			IF fbTimer.Q 
			THEN
				fbTimer(IN := FALSE); 			
				eReadDiagObjState := eCycleDiagObj_Done;
			END_IF

			
		eCycleDiagObj_Done				:	(* Done *)

			eReadDiagObjState := eCycleDiagObj_Init;

			
		eCycleDiagObj_Error			:	(* Error detected *)

			bReadDiagObjError := TRUE;
		
			IF bReadDiagObjReset
			THEN
				bReadDiagObjError 		:= FALSE;
				fbEcCoeSdoRead(bExecute := FALSE);
				eReadDiagObjErrStep 	:= E_TsCycleDiagObj.eCycleDiagObj_NoError;
				eReadDiagObjState 		:= eCycleDiagObj_Init;
			END_IF

	ELSE
		
		eReadDiagObjState := eCycleDiagObj_Init;
		
	END_CASE

	bTempWarning := stSlaveTemp.nInternalTemperature1 >= nWarningLevelTemp1 
						OR stSlaveTemp.nInternalTemperature2 >= nWarningLevelTemp2;

(* End *)
END_ACTION

ACTION act_Signals:
(* Evaluate the input and output signals *)

	IF nEcSlaveState.3 (* Slave in operational state *)
	THEN
	
		(* OP -> transfer the signal states *)
		stSignalStatusMC1.bSafeTorqueOff_STO 					:= stInfoData.nInSafeDataByte1.0;
		stSignalStatusMC1.bSafeSpeedMonitor_SSM_1 				:= stInfoData.nInSafeDataByte1.1;
		stSignalStatusMC1.bSafeSpeedMonitor_SSM_2 				:= stInfoData.nInSafeDataByte1.2;
		stSignalStatusMC1.bSafeOperatingStop_SOS_1	 			:= stInfoData.nInSafeDataByte1.3;
		stSignalStatusMC1.bSafeSpeedRange_SSR_1 				:= stInfoData.nInSafeDataByte1.4;
		stSignalStatusMC1.bSafeDirectionPositive_SDIp 			:= stInfoData.nInSafeDataByte1.5;
		stSignalStatusMC1.bSafeDirectionNegative_SDIn 			:= stInfoData.nInSafeDataByte1.6;
		stSignalStatusMC1.bErrorAcknowledge_ErrAck 				:= stInfoData.nInSafeDataByte1.7;
		stSignalStatusMC1.bNotInUseBit8 						:= stInfoData.nInSafeDataByte2.0;
		stSignalStatusMC1.bNotInUseBit9 						:= stInfoData.nInSafeDataByte2.1;
		stSignalStatusMC1.bNotInUseBit10						:= stInfoData.nInSafeDataByte2.2;
		stSignalStatusMC1.bNotInUseBit11						:= stInfoData.nInSafeDataByte2.3;
		stSignalStatusMC1.bNotInUseBit12						:= stInfoData.nInSafeDataByte2.4;
		stSignalStatusMC1.bNotInUseBit13						:= stInfoData.nInSafeDataByte2.5;
		stSignalStatusMC1.bNotInUseBit14						:= stInfoData.nInSafeDataByte2.6;
		stSignalStatusMC1.bNotInUseBit15						:= stInfoData.nInSafeDataByte2.7;
		
		stSignalStatusMC2.bSafeTorqueOff_STO 					:= stInfoData.nInSafeDataByte3.0;
		stSignalStatusMC2.bSafeSpeedMonitor_SSM_1 				:= stInfoData.nInSafeDataByte3.1;
		stSignalStatusMC2.bSafeSpeedMonitor_SSM_2 				:= stInfoData.nInSafeDataByte3.2;
		stSignalStatusMC2.bSafeOperatingStop_SOS_1 				:= stInfoData.nInSafeDataByte3.3;
		stSignalStatusMC2.bSafeSpeedRange_SSR_1 				:= stInfoData.nInSafeDataByte3.4;
		stSignalStatusMC2.bSafeDirectionPositive_SDIp 			:= stInfoData.nInSafeDataByte3.5;
		stSignalStatusMC2.bSafeDirectionNegative_SDIn		 	:= stInfoData.nInSafeDataByte3.6;
		stSignalStatusMC2.bErrorAcknowledge_ErrAck 				:= stInfoData.nInSafeDataByte3.7;
		stSignalStatusMC2.bNotInUseBit8 						:= stInfoData.nInSafeDataByte4.0;
		stSignalStatusMC2.bNotInUseBit9 						:= stInfoData.nInSafeDataByte4.1;
		stSignalStatusMC2.bNotInUseBit10						:= stInfoData.nInSafeDataByte4.2;
		stSignalStatusMC2.bNotInUseBit11						:= stInfoData.nInSafeDataByte4.3;
		stSignalStatusMC2.bNotInUseBit12						:= stInfoData.nInSafeDataByte4.4;
		stSignalStatusMC2.bNotInUseBit13						:= stInfoData.nInSafeDataByte4.5;
		stSignalStatusMC2.bNotInUseBit14						:= stInfoData.nInSafeDataByte4.6;
		stSignalStatusMC2.bNotInUseBit15						:= stInfoData.nInSafeDataByte4.7;
		
		stSignalControlStatusMC1.bSafeTorqueOff_STO 			:= stInfoData.nOutSafeDataByte1.0;
		stSignalControlStatusMC1.bSafeStop1_SS1_1 				:= stInfoData.nOutSafeDataByte1.1;
		stSignalControlStatusMC1.bSafeStop2_SS2_1 				:= stInfoData.nOutSafeDataByte1.2;
		stSignalControlStatusMC1.bSafeOperatingStop_SOS_1 		:= stInfoData.nOutSafeDataByte1.3;
		stSignalControlStatusMC1.bSafeSpeedRange_SSR_1 			:= stInfoData.nOutSafeDataByte1.4;
		stSignalControlStatusMC1.bSafeDirectionPositive_SDIp 	:= stInfoData.nOutSafeDataByte1.5;
		stSignalControlStatusMC1.bSafeDirectionNegative_SDIn 	:= stInfoData.nOutSafeDataByte1.6;
		stSignalControlStatusMC1.bErrorAcknowledge_ErrAck 		:= stInfoData.nOutSafeDataByte1.7;
		stSignalControlStatusMC1.bNotInUseBit8 					:= stInfoData.nOutSafeDataByte2.0;
		stSignalControlStatusMC1.bNotInUseBit9 					:= stInfoData.nOutSafeDataByte2.1;
		stSignalControlStatusMC1.bNotInUseBit10					:= stInfoData.nOutSafeDataByte2.2;
		stSignalControlStatusMC1.bNotInUseBit11					:= stInfoData.nOutSafeDataByte2.3;
		stSignalControlStatusMC1.bNotInUseBit12					:= stInfoData.nOutSafeDataByte2.4;
		stSignalControlStatusMC1.bNotInUseBit13					:= stInfoData.nOutSafeDataByte2.5;
		stSignalControlStatusMC1.bNotInUseBit14					:= stInfoData.nOutSafeDataByte2.6;
		stSignalControlStatusMC1.bNotInUseBit15					:= stInfoData.nOutSafeDataByte2.7;

		stSignalControlStatusMC2.bSafeTorqueOff_STO 			:= stInfoData.nOutSafeDataByte3.0;
		stSignalControlStatusMC2.bSafeStop1_SS1_1 				:= stInfoData.nOutSafeDataByte3.1;
		stSignalControlStatusMC2.bSafeStop2_SS2_1 				:= stInfoData.nOutSafeDataByte3.2;
		stSignalControlStatusMC2.bSafeOperatingStop_SOS_1 		:= stInfoData.nOutSafeDataByte3.3;
		stSignalControlStatusMC2.bSafeSpeedRange_SSR_1 			:= stInfoData.nOutSafeDataByte3.4;
		stSignalControlStatusMC2.bSafeDirectionPositive_SDIp 	:= stInfoData.nOutSafeDataByte3.5;
		stSignalControlStatusMC2.bSafeDirectionNegative_SDIn 	:= stInfoData.nOutSafeDataByte3.6;
		stSignalControlStatusMC2.bErrorAcknowledge_ErrAck 		:= stInfoData.nOutSafeDataByte3.7;
		stSignalControlStatusMC2.bNotInUseBit8 					:= stInfoData.nOutSafeDataByte4.0;
		stSignalControlStatusMC2.bNotInUseBit9 					:= stInfoData.nOutSafeDataByte4.1;
		stSignalControlStatusMC2.bNotInUseBit10					:= stInfoData.nOutSafeDataByte4.2;
		stSignalControlStatusMC2.bNotInUseBit11					:= stInfoData.nOutSafeDataByte4.3;
		stSignalControlStatusMC2.bNotInUseBit12					:= stInfoData.nOutSafeDataByte4.4;
		stSignalControlStatusMC2.bNotInUseBit13					:= stInfoData.nOutSafeDataByte4.5;
		stSignalControlStatusMC2.bNotInUseBit14					:= stInfoData.nOutSafeDataByte4.6;
		stSignalControlStatusMC2.bNotInUseBit15					:= stInfoData.nOutSafeDataByte4.7;
		
	ELSE
		
		(* Error -> clear the signal states *)
		stSignalStatusMC1.bSafeTorqueOff_STO 					:= FALSE;
		stSignalStatusMC1.bSafeSpeedMonitor_SSM_1 				:= FALSE;
		stSignalStatusMC1.bSafeSpeedMonitor_SSM_2 				:= FALSE;
		stSignalStatusMC1.bSafeOperatingStop_SOS_1	 			:= FALSE;
		stSignalStatusMC1.bSafeSpeedRange_SSR_1 				:= FALSE;
		stSignalStatusMC1.bSafeDirectionPositive_SDIp 			:= FALSE;
		stSignalStatusMC1.bSafeDirectionNegative_SDIn 			:= FALSE;
		stSignalStatusMC1.bErrorAcknowledge_ErrAck 				:= FALSE;
		stSignalStatusMC1.bNotInUseBit8 						:= FALSE;
		stSignalStatusMC1.bNotInUseBit9 						:= FALSE;
		stSignalStatusMC1.bNotInUseBit10						:= FALSE;
		stSignalStatusMC1.bNotInUseBit11						:= FALSE;
		stSignalStatusMC1.bNotInUseBit12						:= FALSE;
		stSignalStatusMC1.bNotInUseBit13						:= FALSE;
		stSignalStatusMC1.bNotInUseBit14						:= FALSE;
		stSignalStatusMC1.bNotInUseBit15						:= FALSE;
		
		stSignalStatusMC2.bSafeTorqueOff_STO 					:= FALSE;
		stSignalStatusMC2.bSafeSpeedMonitor_SSM_1 				:= FALSE;
		stSignalStatusMC2.bSafeSpeedMonitor_SSM_2 				:= FALSE;
		stSignalStatusMC2.bSafeOperatingStop_SOS_1 				:= FALSE;
		stSignalStatusMC2.bSafeSpeedRange_SSR_1 				:= FALSE;
		stSignalStatusMC2.bSafeDirectionPositive_SDIp 			:= FALSE;
		stSignalStatusMC2.bSafeDirectionNegative_SDIn		 	:= FALSE;
		stSignalStatusMC2.bErrorAcknowledge_ErrAck 				:= FALSE;
		stSignalStatusMC2.bNotInUseBit8 						:= FALSE;
		stSignalStatusMC2.bNotInUseBit9 						:= FALSE;
		stSignalStatusMC2.bNotInUseBit10						:= FALSE;
		stSignalStatusMC2.bNotInUseBit11						:= FALSE;
		stSignalStatusMC2.bNotInUseBit12						:= FALSE;
		stSignalStatusMC2.bNotInUseBit13						:= FALSE;
		stSignalStatusMC2.bNotInUseBit14						:= FALSE;
		stSignalStatusMC2.bNotInUseBit15						:= FALSE;
		
		stSignalControlStatusMC1.bSafeTorqueOff_STO 			:= FALSE;
		stSignalControlStatusMC1.bSafeStop1_SS1_1 				:= FALSE;
		stSignalControlStatusMC1.bSafeStop2_SS2_1 				:= FALSE;
		stSignalControlStatusMC1.bSafeOperatingStop_SOS_1 		:= FALSE;
		stSignalControlStatusMC1.bSafeSpeedRange_SSR_1 			:= FALSE;
		stSignalControlStatusMC1.bSafeDirectionPositive_SDIp 	:= FALSE;
		stSignalControlStatusMC1.bSafeDirectionNegative_SDIn 	:= FALSE;
		stSignalControlStatusMC1.bErrorAcknowledge_ErrAck 		:= FALSE;
		stSignalControlStatusMC1.bNotInUseBit8 					:= FALSE;
		stSignalControlStatusMC1.bNotInUseBit9 					:= FALSE;
		stSignalControlStatusMC1.bNotInUseBit10					:= FALSE;
		stSignalControlStatusMC1.bNotInUseBit11					:= FALSE;
		stSignalControlStatusMC1.bNotInUseBit12					:= FALSE;
		stSignalControlStatusMC1.bNotInUseBit13					:= FALSE;
		stSignalControlStatusMC1.bNotInUseBit14					:= FALSE;
		stSignalControlStatusMC1.bNotInUseBit15					:= FALSE;

		stSignalControlStatusMC2.bSafeTorqueOff_STO 			:= FALSE;
		stSignalControlStatusMC2.bSafeStop1_SS1_1 				:= FALSE;
		stSignalControlStatusMC2.bSafeStop2_SS2_1 				:= FALSE;
		stSignalControlStatusMC2.bSafeOperatingStop_SOS_1 		:= FALSE;
		stSignalControlStatusMC2.bSafeSpeedRange_SSR_1 			:= FALSE;
		stSignalControlStatusMC2.bSafeDirectionPositive_SDIp 	:= FALSE;
		stSignalControlStatusMC2.bSafeDirectionNegative_SDIn 	:= FALSE;
		stSignalControlStatusMC2.bErrorAcknowledge_ErrAck 		:= FALSE;
		stSignalControlStatusMC2.bNotInUseBit8 					:= FALSE;
		stSignalControlStatusMC2.bNotInUseBit9 					:= FALSE;
		stSignalControlStatusMC2.bNotInUseBit10					:= FALSE;
		stSignalControlStatusMC2.bNotInUseBit11					:= FALSE;
		stSignalControlStatusMC2.bNotInUseBit12					:= FALSE;
		stSignalControlStatusMC2.bNotInUseBit13					:= FALSE;
		stSignalControlStatusMC2.bNotInUseBit14					:= FALSE;
		stSignalControlStatusMC2.bNotInUseBit15					:= FALSE;

	END_IF

(* End *)
END_ACTION

END_FUNCTION_BLOCK

// ---- POUs/Motion/NCI.TcPOU
PROGRAM NCI
VAR
(* NCI G code stuff *)

	in_stItpToPlc		AT 	%I*:	NCTOPLC_NCICHANNEL_REF;
	out_stPlcToItp		AT	%Q*:	PLCTONC_NCICHANNEL_REF;
	
	bRunNCI				: BOOL;
	bErrorAck			: BOOL;

(*
	g_strProgram:	STRING := 'Hard Disk2\TestIt.nc';	(* USB stick with CE OS *)
*)
	g_strProgram		: STRING := 'C:\btest.nc';

	bNCIExec			: BOOL;
	bNCIBusy			: BOOL := FALSE;
	bNciErr				: BOOL := FALSE;
	nNciErrId			: UDINT := 0;

	nNCI_State			: UDINT := 0;
	nLastState			: UDINT	:= 0;	(* for debugging purposes *)
	fbBuildGrp			: CfgBuildExt3DGroup;
	fbLoadProg			: ItpLoadProgEx;
	fbStart				: ItpStartStopEx;
	
	fbConfirm			: ItpConfirmHsk;
	bConfirm			: BOOL := FALSE;
	
	fbClearGrp			: CfgReconfigGroup;
	fbResetItp			: ItpResetEx2;
	nItpState			: UDINT;

	bPenDown : BOOL;

	fbADSREAD_NciLine	: ADSREAD;
	sGCodeLine			: STRING(254);
	sGCodeLineLast		: STRING(254);
	bReadGcodeLine		: BOOL;
	bItpReset			: BOOL;

	aGCodeLines			: ARRAY[0..9] OF STRING[254];
	iLine				: UINT;
END_VAR

ItpSetOverridePercent(100.0, out_stPlcToItp);

CASE nNCI_State OF
0:
	if bRunNCI then
		nNCI_State := 5;
	END_IF
	
5:
	bNCIBusy	:= TRUE;
	bNciErr	:= FALSE;
	nNciErrId	:= 0;
	nLastState	:= 0;
	nNCI_State 	:= 10;
	FOR iLine := 0 TO 9 DO
			aGCodeLines[iLine]:='';
	END_FOR


10:
	(* build interpolation group *)
	fbBuildGrp(
		bExecute	:= TRUE ,
		nGroupId	:= ItpGetGroupId(sNciToPlc:=in_stItpToPlc),
		nXAxisId	:= stAxis3.NcToPlc.AxisId,
		nYAxisId	:= stAxis4.NcToPlc.AxisId,
		nZAxisId	:= 0,
		nQ1AxisId:= 0,
		nQ2AxisId:= 0,
		nQ3AxisId:= 0,
		nQ4AxisId:= 0,
		nQ5AxisId:= 0,
		tTimeOut:= T#200ms);

	IF NOT fbBuildGrp.bBusy THEN
		fbBuildGrp( bExecute := FALSE );
		IF NOT fbBuildGrp.bErr THEN
			nNCI_State	:= 20;
		ELSE
			(* an error occured *)
			bNciErr		:= TRUE;
			nNciErrId	:= fbBuildGrp.nErrId;
			nLastState	:= nNCI_State;
			nNCI_State	:= 9999;
		END_IF
	END_IF

20:
	(* load part program *)
	fbLoadProg(
		bExecute	:= TRUE,
		sPrg		:= g_strProgram,
		nLength		:= INT_TO_UDINT(LEN(g_strProgram)),
		tTimeOut	:= t#200ms,
		sNciToPlc:= in_stItpToPlc );

	IF NOT fbLoadProg.bBusy THEN
		fbLoadProg( bExecute:=FALSE, sNciToPlc:=in_stItpToPlc );
		IF NOT fbLoadProg.bErr THEN
			nNCI_State	:= 30;
		ELSE
			(* an error occured *)
			bNciErr		:= TRUE;
			nNciErrId	:= fbLoadProg.nErrId;
			nLastState	:= nNCI_State;
			nNCI_State	:= 9999;
		END_IF
	END_IF

30:
	(* wait until interpreter is in ready state *)
	nItpState	:=	ItpGetStateInterpreter( in_stItpToPlc );
	IF nItpState = NCI_INTERPRETER_READY THEN
		(* load part program succeeded *)
		nNCI_State	:= 40;
	ELSIF nItpState = NCI_INTERPRETER_ABORTED THEN
		(* load program failed - probably there is a load time error, e.g. syntax error *)
		(* add error handling here *)
		bNciErr		:= TRUE;
		nNciErrId	:= 4711;	(* substitute with own error code *)
		nLastState	:= nNCI_State;
		nNCI_State	:= 9999;
	END_IF

40:
	(* start part program *)
	fbStart(
		bStart	:= TRUE,
		bStop		:= FALSE,
		tTimeOut	:= t#200ms,
		sNciToPlc:= in_stItpToPlc );

	IF NOT fbStart.bBusy THEN
		fbStart( bStart:=FALSE, sNciToPlc:=in_stItpToPlc );
		IF NOT fbStart.bErr THEN
			nNCI_State	:= 50;
		ELSE
			(* an error occured *)
			bNciErr		:= TRUE;
			nNciErrId	:= fbStart.nErrId;
			nLastState	:= nNCI_State;
			nNCI_State	:= 9999;
		END_IF
	END_IF

50:
	(* check if the part program is really started *)
	(* as long as the part program is active we are not in the ready state *)
	(* if the part program has finished without an error we switch back to the ready state *)
	(* if the program has finished with an error the interpreter is in the aborted state *)
	nItpState	:=	ItpGetStateInterpreter( in_stItpToPlc );
	IF nItpState <> NCI_INTERPRETER_READY THEN
		nNCI_State	:= 60;
		// bReadGcodeLine := TRUE;
	END_IF

60:
	(* Confirmed m-functions *)
	(*
	IF ( ItpIsHskMFunc(in_stItpToPlc) ) THEN
		bConfirm	:= TRUE;
	ELSE
		bConfirm	:= FALSE;
	END_IF

	fbConfirm(
		bExecute:= bConfirm,
		sNciToPlc:= in_stItpToPlc,
		sPlcToNci:= out_stPlcToItp );

	IF NOT fbConfirm.bBusy THEN
		IF fbConfirm.bErr THEN
			(* an error occured *)
			(* this usually can just occur, if a confirmation is triggered without a request *)
			bNCIErr		:= TRUE;
			iNCIErrId	:= fbStart.nErrId;
			iNCILastState	:= iNCIState;
			iNCIState	:= 9999;
		END_IF
	END_IF
	*)

(* code for fast M function with no handshaking - example M100/M101 to trigger 'Pen down' boolean *)
	IF ItpIsFastMFunc(100, in_stItpToPlc ) THEN
		bPenDown:= TRUE;
	ELSE
		bPenDown:= FALSE;
	END_IF

	nItpState	:=	ItpGetStateInterpreter( in_stItpToPlc );
	IF nItpState = NCI_INTERPRETER_READY THEN
		(* part program is finished without an error *)
		nNCI_State	:= 70;
	ELSIF nItpState = NCI_INTERPRETER_ABORTED THEN
		(* a runtime error occured - e.g. a lag distance error occured *)
		bNciErr		:= TRUE;
		nNciErrId	:= ItpGetError(in_stItpToPlc);
		nLastState	:= nNCI_State;
		nNCI_State	:= 9999;
	END_IF

	(* Read executing Gcode lines *)
	fbADSREAD_NciLine(
		NETID:= '',
		PORT:= 500,
		IDXGRP:= 16#2302,
		IDXOFFS:= 16#20000001,
		LEN:= 248,
		DESTADDR:= ADR(sGCodeLine),
		READ:= bReadGcodeLine,
		TMOUT:= t#200ms,
		BUSY=> ,
		ERR=> ,
		ERRID=> );

	IF fbADSREAD_NciLine.BUSY = FALSE THEN
		IF bReadGcodeLine = TRUE THEN
			bReadGcodeLine:=FALSE;
			IF sGCodeLineLast<>sGCodeLine THEN
				// shift table down and add line to top of table
				MEMMOVE(destAddr:= ADR(aGCodeLines[1]), srcAddr:= ADR(aGCodeLines[0]), n:= 254*9);
				aGCodeLines[0]:=sGCodeLine;
				sGCodeLineLast:=sGCodeLine;
			END_IF
		ELSE
			bReadGcodeLine:=TRUE;
		END_IF
	END_IF

70:
	(* clear interpolation group *)
	fbClearGrp(
		bExecute:= TRUE,
		nGroupId:= ItpGetGroupId(sNciToPlc:=in_stItpToPlc),
		tTimeOut:= T#200ms);

	IF NOT fbClearGrp.bBusy THEN
		fbClearGrp(bExecute:= FALSE);
		IF NOT fbClearGrp.bErr THEN
			nNCI_State	:= 100;
		ELSE
			(* an error occured *)
			bNciErr		:= TRUE;
			nNciErrId	:= fbClearGrp.nErrId;
			nLastState	:= nNCI_State;
			nNCI_State	:= 9999;
		END_IF
	END_IF

100:	(* Finished NCI successfully *)
	bNciBusy	:= FALSE;
	fbBuildGrp( bExecute:=FALSE );
	fbLoadProg( bExecute:=FALSE, sNciToPlc:=in_stItpToPlc );
	fbStart( bStart:=FALSE, bStop:=FALSE, sNciToPlc:=in_stItpToPlc );
	fbClearGrp(bExecute:= FALSE);

	bPenDown:= FALSE;
	bReadGcodeLine:=FALSE;

	nNci_State	:= 0;

9999:
	bNCIBusy	:= FALSE;
	fbBuildGrp( bExecute:=FALSE );
	fbLoadProg( bExecute:=FALSE, sNciToPlc:=in_stItpToPlc );
	fbStart( bStart:=FALSE, bStop:=FALSE, sNciToPlc:=in_stItpToPlc );
	fbClearGrp(bExecute:= FALSE);

	bPenDown:= FALSE;
	bReadGcodeLine:=FALSE;

	IF bErrorAck THEN
		nNCI_State	:= 0;
		nNciErrId	:= 0;
	END_IF

END_CASE

END_PROGRAM

// ---- POUs/Motion/CamTable.TcPOU
PROGRAM CamTable
VAR
	bLoadPoints: BOOL;
	bCamInit			: BOOL;

	arCamTable			: ARRAY [0..iNumPts, 0..1] OF LREAL;
	CamTblSelect		: MC_CamTableSelect;
	CamTableRef			: MC_Cam_Ref;
	ST_CamInOptions_V2	: ST_CamInOptions_V2;

	CamIn_v2			: MC_CamIn_V2;
	CamOut				: MC_CamOut;
	bCamIn				: BOOL;

	osrTblSlct			: F_TRIG;
	bPeriodic			: BOOL;

	iInterpType			: UINT :=1;		// start with spline

	iSelX				: INT;			// selected visualization col
	iSelY				: INT;			// selected visualization row 
	
END_VAR

VAR CONSTANT
	iNumPts 			: UDINT := 5;
END_VAR

Cam_Setup();

IF bLoadPoints THEN
	LoadPoints();
	bLoadPoints:=FALSE;
END_IF

IF bCamInit THEN
	Cam_Init();
	bCamInit := FALSE;
END_IF

ACTION Cam_Init:

CamTableRef.pArray := ADR(arCamTable);
CamTableRef.ArraySize := SIZEOF(arCamTable);

CamTableRef.TableType := MC_TABLETYPE_EQUIDISTANT ;

CamTableRef.NoOfRows := iNumPts;
CamTableRef.NoOfColumns := 2;
ST_CamInOptions_V2.CamOperationMode:=CAMOPERATIONMODE_ADDITIVE;


CASE iInterpType OF
0:
	ST_CamInOptions_V2.InterpolationType:=MC_INTERPOLATIONTYPE_LINEAR;
1:
	ST_CamInOptions_V2.InterpolationType:=MC_INTERPOLATIONTYPE_SPLINE;
2:
	ST_CamInOptions_V2.InterpolationType:=MC_INTERPOLATIONTYPE_SLIDINGSPLINE;
END_CASE
END_ACTION

ACTION Cam_Setup:
osrTblSlct(CLK := bCamInit); // F_TRIG
CamIn_v2(
    Master := stAxis3,
    Slave := stAxis4,
    Execute := bCamIn,
    ActivationMode := MC_CAMACTIVATION_INSTANTANEOUS,
    CamTableID := 2,
    Options := ST_CamInOptions_V2); // MC_CamIn_V2
CamTblSelect(
    Execute := NOT CamTblSelect.Done AND osrTblSlct.Q,
    Periodic := bPeriodic,
    CamTableID := 2,
    Master := stAxis3,
    Slave := stAxis4,
    CamTable := CamTableRef); // MC_CamTableSelect
CamOut(Execute := NOT(bCamIn), Slave := stAxis4); // MC_CamOut
END_ACTION

ACTION LoadPoints:
arCamTable[0,0] := 0;
arCamTable[0,1] := 0;

arCamTable[1,0] := 250;
arCamTable[1,1] := 500;

arCamTable[2,0] := 500;
arCamTable[2,1] := 1000;

arCamTable[3,0] := 750;
arCamTable[3,1] := 500;

arCamTable[4,0] := 1000;
arCamTable[4,1] := 0;
END_ACTION

END_PROGRAM

// ---- POUs/Motion/Ext_SP_Gen.TcPOU
PROGRAM Ext_SP_Gen
VAR
	bMstrExtSP			: BOOL;
	ExtSP_Enable		: MC_ExtSetPointGenEnable;
	ExtSP_Disable		: MC_ExtSetPointGenDisable;	

	lrPosCmd			: LREAL;
	lrVeloCmd			: LREAL;
	lrAccelCmd			: LREAL;

	rDeg				: REAL;
	rDegStep			: REAL := 0.1;
	lrSinWave			: LREAL;
	rSinAmp				: REAL := 30.0;
	
	bSinGen				: BOOL;
	bAddSin				: BOOL;

	diDir: DINT := 1;
	
	lrPosInput: LREAL;
END_VAR

IF bSinGen THEN
	rDeg:=rDeg+rDegStep;
	IF rDeg >= 360.0 THEN
		rDeg:=0.0;
	END_IF
END_IF

lrSinWave:=rSinAmp*SIN(rDeg*3.14159/180.0);	// SIN function uses radian input

IF bAddSin THEN
	lrPosCmd:=lrPosInput+lrSinWave;
ELSE
	lrPosCmd:=lrPosInput;
END_IF

MC_ExtSetPointGenFeed(
	lrPosCmd,
	lrVeloCmd,
	lrAccelCmd,
	diDir,
	stAxis3);

ExtSP_Enable(
	Axis:= stAxis3, 
	Execute:= bMstrExtSP, 
	Position:= , 
	PositionType:= POSITIONTYPE_ABSOLUTE, 
	Done=> , 
	Busy=> , 
	Error=> , 
	ErrorID=> , 
	Enabled=> );
	
ExtSP_Disable(
	Axis:= stAxis3, 
	Execute:= NOT(bMstrExtSP), 
	Done=> , 
	Busy=> , 
	Error=> , 
	ErrorID=> , 
	Enabled=> );

END_PROGRAM

// ---- POUs/SampleIEC Languages/MAIN_CFC.TcPOU
PROGRAM MAIN_CFC
VAR
	Timer			: TON;
	fbCFC_SamplePOU : FB_CFC_SamplePOU;

	eOperation		: E_Operation := eOp_Add;
	eOperationPrev	: E_Operation := eOp_Add;
	iResultC		: DINT;
	bZero			: BOOL;
	bPos			: BOOL;
	bNeg			: BOOL;
	bTest			: BOOL;
	tTimerValue		: TIME := T#3S;
END_VAR
VAR // added by the converter: edge detectors and wires of the graphical bodies
    _w1, _w2, _w3 : E_Operation;
END_VAR

bTest := (bZero AND bPos OR bPos XOR bNeg) AND iResultC <= 0 AND Timer.ET > T#500ms OR Timer.ET <= T#500ms;
// Timer
Timer(IN := NOT Timer.Q, PT := tTimerValue); // TON
IF NOT Timer.Q THEN JMP CALLFB; END_IF
// State machine
_w1 := SEL(eOp_Add = eOperation AND Timer.Q, eOperation, eOp_Mul);
eOperation := _w1;
IF _w1 <> eOperationPrev AND _w1 = eOp_Mul THEN JMP CallFB; END_IF
_w2 := SEL(eOp_Sub = eOperation AND Timer.Q, eOperation, eOp_Add);
eOperation := _w2;
IF _w2 <> eOperationPrev AND _w2 = eOp_Add THEN JMP CallFB; END_IF
_w3 := SEL(eOp_Mul = eOperation AND Timer.Q, eOperation, eOp_Sub);
eOperation := _w3;
IF _w3 <> eOperationPrev AND _w3 = eOp_Sub THEN JMP CallFB; END_IF
// FB Call
CallFB: ;
eOperationPrev := eOperation;
fbCFC_SamplePOU(eOperation := eOperation); // FB_CFC_SamplePOU
iResultC := fbCFC_SamplePOU.iResultC;
bZero := fbCFC_SamplePOU.iResultC = 0;
bPos := fbCFC_SamplePOU.iResultC > 0;
bNeg := fbCFC_SamplePOU.iResultC < 0;

END_PROGRAM

// ---- POUs/SampleIEC Languages/FunctionBlocks/FB_CFC_SamplePOU.TcPOU
FUNCTION_BLOCK FB_CFC_SamplePOU
VAR_INPUT
//	eOperation	: INT;
	eOperation	: E_Operation;
END_VAR
VAR_OUTPUT
	iResultC	: DINT;
END_VAR
VAR
	arrDataA	: ARRAY [1..iMax] OF DINT;
	arrDataB	: ARRAY [1..iMax] OF DINT;
	arrDataC	: ARRAY [1..iMax] OF DINT;
	I 			: DINT;
	bInit		: BOOL := TRUE;
END_VAR
VAR CONSTANT
	iMax 		: DINT := 10;
END_VAR
VAR // added by the converter: edge detectors and wires of the graphical bodies
    _w1, _w2, _w4, _w6, _w9 : DINT;
    _w3, _w5, _w8 : ANY;
    _w7 : BOOL;
END_VAR

IF NOT bInit THEN JMP SkipInit; END_IF
bInit := FALSE;
I := 1;
Init: ;
_w1 := iMax - I;
arrDataA[I] := _w1;
arrDataB[I] := _w1 + 1;
_w2 := I + 1;
I := _w2;
IF _w2 <= iMax THEN JMP Init; END_IF
SkipInit: ;
IF eOperation = eOp_Add THEN JMP OP_Add; END_IF
IF eOperation = eOp_Sub THEN JMP OP_Sub; END_IF
IF eOperation = eOp_Mul THEN JMP OP_Mul; END_IF
IF TRUE THEN JMP END; END_IF
OP_Add: ;
iResultC := 0;
I := 1 + 0;
WHILE4_0: ;
IF I > iMax THEN JMP END; END_IF
_w3 := arrDataA[I] + arrDataB[I];
arrDataC[I] := _w3;
iResultC := iResultC + _w3;
_w4 := I + 1;
I := _w4;
IF _w4 >= _w4 THEN JMP WHILE4_0; END_IF
OP_Sub: ;
iResultC := 0;
I := 1 + 0;
Repeat5_0: ;
_w5 := arrDataA[I] - arrDataB[I];
arrDataC[I] := _w5;
iResultC := iResultC + _w5 * -1;
_w6 := I + 1;
I := _w6;
_w7 := _w6 <= iMax;
IF _w7 THEN JMP Repeat5_0; END_IF
IF _w7 = FALSE THEN JMP END; END_IF
OP_Mul: ;
I := 1;
iResultC := 1;
FOR6_0: ;
IF I > iMax THEN JMP END; END_IF
_w8 := arrDataA[I] * arrDataB[I];
arrDataC[I] := _w8;
iResultC := iResultC * _w8;
_w9 := I + 1;
I := _w9;
IF _w9 <= iMax THEN JMP FOR6_0; END_IF
END: ;

END_FUNCTION_BLOCK

// ---- POUs/SampleIEC Languages/MAIN_CFC_PageOriented.TcPOU
PROGRAM MAIN_CFC_PageOriented
VAR
	Timer			: TON;
	fbCFC_SamplePOUPageOriented : FB_CFC_SamplePOUPageOriented;

	eOperation		: E_Operation := eOp_Add;
	eOperationPrev	: E_Operation := eOp_Add;
	iResultC		: DINT;
	bZero			: BOOL;
	bPos			: BOOL;
	bNeg			: BOOL;
	bTest			: BOOL;
	tTimerValue		: TIME := T#3S;
END_VAR
VAR // added by the converter: edge detectors and wires of the graphical bodies
    _w1, _w2, _w3 : E_Operation;
END_VAR


// PAGE Test Test Signal
bTest := (bZero AND bPos OR bPos XOR bNeg) AND iResultC <= 0 AND Timer.ET > T#500ms OR Timer.ET <= T#500ms;

// PAGE Timer
// Timer
Timer(IN := NOT Timer.Q, PT := tTimerValue); // TON
IF NOT Timer.Q THEN JMP CALLFB; END_IF

// PAGE State Machine State Machine and FB Call
// State machine
_w1 := SEL(eOp_Add = eOperation AND Timer.Q, eOperation, eOp_Mul);
eOperation := _w1;
IF _w1 <> eOperationPrev AND _w1 = eOp_Mul THEN JMP CallFB; END_IF
_w2 := SEL(eOp_Sub = eOperation AND Timer.Q, eOperation, eOp_Add);
eOperation := _w2;
IF _w2 <> eOperationPrev AND _w2 = eOp_Add THEN JMP CallFB; END_IF
_w3 := SEL(eOp_Mul = eOperation AND Timer.Q, eOperation, eOp_Sub);
eOperation := _w3;
IF _w3 <> eOperationPrev AND _w3 = eOp_Sub THEN JMP CallFB; END_IF

// PAGE Call FB Function Block Call
// FB Call
CallFB: ;
fbCFC_SamplePOUPageOriented(eOperation := eOperation); // FB_CFC_SamplePouPageOriented
iResultC := fbCFC_SamplePOUPageOriented.iResultC;
eOperationPrev := eOperation;
bZero := fbCFC_SamplePOUPageOriented.iResultC = 0;
bPos := fbCFC_SamplePOUPageOriented.iResultC > 0;
bNeg := fbCFC_SamplePOUPageOriented.iResultC < 0;

END_PROGRAM

// ---- POUs/SampleIEC Languages/FunctionBlocks/FB_CFC_SamplePouPageOriented.TcPOU
FUNCTION_BLOCK FB_CFC_SamplePouPageOriented
VAR_INPUT
//	eOperation	: INT;
	eOperation	: E_Operation;
END_VAR
VAR_OUTPUT
	iResultC	: DINT;
END_VAR
VAR
	arrDataA	: ARRAY [1..iMax] OF DINT;
	arrDataB	: ARRAY [1..iMax] OF DINT;
	arrDataC	: ARRAY [1..iMax] OF DINT;
	I 			: DINT;
	bInit		: BOOL := TRUE;
END_VAR
VAR CONSTANT
	iMax 		: DINT := 10;
END_VAR
VAR // added by the converter: edge detectors and wires of the graphical bodies
    _w1, _w2, _w4, _w6, _w10 : DINT;
    _w3, _w5, _w9 : ANY;
    _w7, _w8 : BOOL;
END_VAR


// PAGE Init Initialization
IF NOT bInit THEN JMP SkipInit; END_IF
bInit := FALSE;
I := 1;
Init: ;
_w1 := iMax - I;
arrDataB[I] := _w1 + 1;
arrDataA[I] := _w1;
_w2 := I + 1;
I := _w2;
IF _w2 <= iMax THEN JMP Init; END_IF
SkipInit: ;
IF eOperation = eOp_Add THEN JMP OP_Add; END_IF
IF eOperation = eOp_Sub THEN JMP OP_Sub; END_IF
IF eOperation = eOp_Mul THEN JMP OP_Mul; END_IF
IF TRUE THEN JMP END; END_IF

// PAGE Add Operation Add
OP_Add: ;
I := 1 + 0;
iResultC := 0;
WHILE4_0: ;
IF I > iMax THEN JMP END; END_IF
_w3 := arrDataA[I] + arrDataB[I];
iResultC := iResultC + _w3;
arrDataC[I] := _w3;
_w4 := I + 1;
I := _w4;
IF _w4 >= _w4 THEN JMP WHILE4_0; END_IF

// PAGE Sub Operation Sub
OP_Sub: ;
I := 1 + 0;
iResultC := 0;
Repeat5_0: ;
_w5 := arrDataA[I] - arrDataB[I];
arrDataC[I] := _w5;
iResultC := iResultC + _w5 * -1;
_w6 := I + 1;
I := _w6;
_w7 := _w6 <= iMax;
_w8 := _w7 = FALSE;
IF _w7 THEN JMP Repeat5_0; END_IF
IF _w8 THEN JMP END; END_IF

// PAGE Mul Operation Mul
OP_Mul: ;
I := 1;
iResultC := 1;
FOR6_0: ;
IF I > iMax THEN JMP END; END_IF
_w9 := arrDataA[I] * arrDataB[I];
iResultC := iResultC * _w9;
arrDataC[I] := _w9;
_w10 := I + 1;
I := _w10;
IF _w10 <= iMax THEN JMP FOR6_0; END_IF
END: ;

END_FUNCTION_BLOCK

// ---- POUs/SampleIEC Languages/MAIN_FBD_IL_LD.TcPOU
PROGRAM MAIN_FBD_IL_LD //use menu "FBD/IL/LD" to switch language between FBD, IL and LD offline or online 
VAR
	Timer					: TON;
	fbFBD_IL_LD_SamplePOU 	: FB_FBD_IL_LD_SamplePOU;

	eOperation		: E_Operation := eOp_Add;
	eOperationPrev	: E_Operation := eOp_Add;
	iResultC		: DINT;
	bZero			: BOOL;
	bPos			: BOOL;
	bNeg			: BOOL;
	bTest			: BOOL;
	tTimerValue		: TIME := T#3S;
END_VAR
VAR // added by the converter: edge detectors and wires of the graphical bodies
    _w1, _w2, _w3 : ANY;
END_VAR

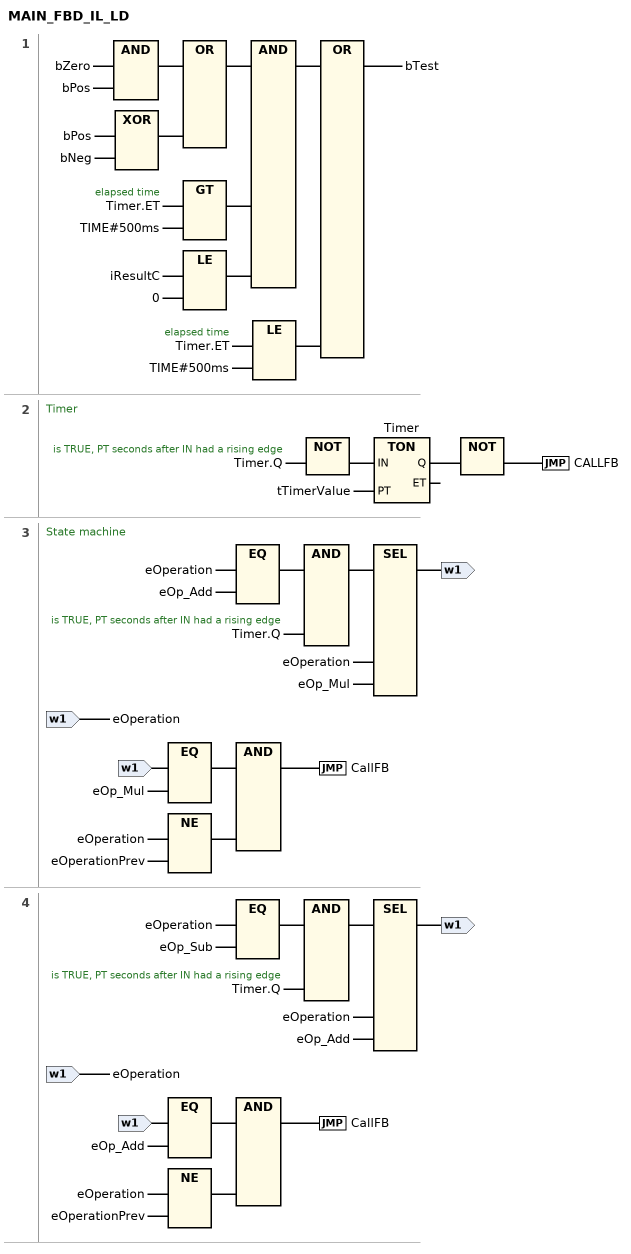
// NETWORK 1
//   Timer.ET: elapsed time
bTest := (bZero AND bPos OR bPos XOR bNeg) AND Timer.ET > TIME#500ms AND iResultC <= 0 OR Timer.ET <= TIME#500ms;

// NETWORK 2
//  Timer
//   Timer.Q: is TRUE, PT seconds after IN had a rising edge
Timer(IN := NOT Timer.Q, PT := tTimerValue); // TON
IF NOT Timer.Q THEN JMP CALLFB; END_IF

// NETWORK 3
//  State machine
//   Timer.Q: is TRUE, PT seconds after IN had a rising edge
_w1 := SEL(eOperation = eOp_Add AND Timer.Q, eOperation, eOp_Mul);
eOperation := _w1;
IF _w1 = eOp_Mul AND eOperation <> eOperationPrev THEN JMP CallFB; END_IF

// NETWORK 4
//   Timer.Q: is TRUE, PT seconds after IN had a rising edge
_w2 := SEL(eOperation = eOp_Sub AND Timer.Q, eOperation, eOp_Add);
eOperation := _w2;
IF _w2 = eOp_Add AND eOperation <> eOperationPrev THEN JMP CallFB; END_IF

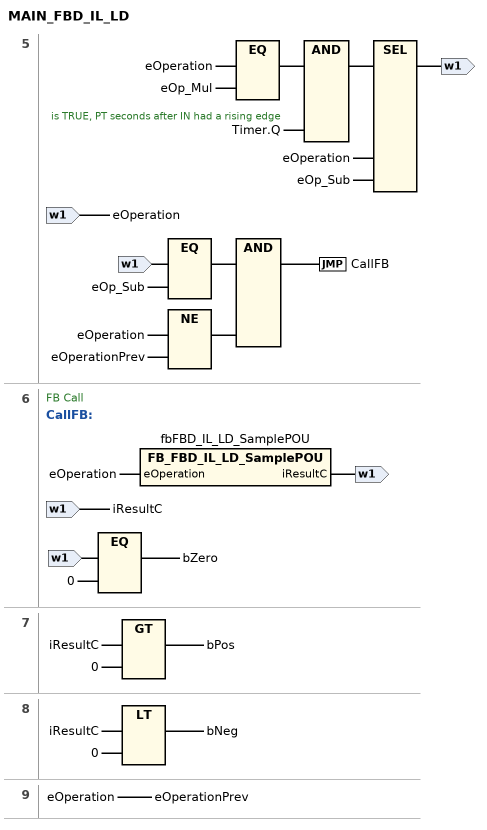
// NETWORK 5
//   Timer.Q: is TRUE, PT seconds after IN had a rising edge
_w3 := SEL(eOperation = eOp_Mul AND Timer.Q, eOperation, eOp_Sub);
eOperation := _w3;
IF _w3 = eOp_Sub AND eOperation <> eOperationPrev THEN JMP CallFB; END_IF

// NETWORK 6
//  FB Call
CallFB:
fbFBD_IL_LD_SamplePOU(eOperation := eOperation); // FB_FBD_IL_LD_SamplePOU
iResultC := fbFBD_IL_LD_SamplePOU.iResultC;
bZero := fbFBD_IL_LD_SamplePOU.iResultC = 0;

// NETWORK 7
bPos := iResultC > 0;

// NETWORK 8
bNeg := iResultC < 0;

// NETWORK 9
eOperationPrev := eOperation;

END_PROGRAM

// ---- POUs/SampleIEC Languages/FunctionBlocks/FB_FBD_IL_LD_SamplePOU.TcPOU
FUNCTION_BLOCK FB_FBD_IL_LD_SamplePOU
VAR_INPUT
//	eOperation	: INT;
	eOperation	: E_Operation;
END_VAR
VAR_OUTPUT
	iResultC	: DINT;
END_VAR
VAR
	arrDataA	: ARRAY [1..iMax] OF DINT;
	arrDataB	: ARRAY [1..iMax] OF DINT;
	arrDataC	: ARRAY [1..iMax] OF DINT;
	I 			: DINT;
	bInit		: BOOL := TRUE;
	bEnd		: BOOL;
	bRepeat		: BOOL;
	bAtTheEnd	: BOOL;
END_VAR
VAR CONSTANT
	iMax 		: DINT := 10;
END_VAR
VAR // added by the converter: edge detectors and wires of the graphical bodies
    _w1, _w2, _w3, _w4, _w5, _w6, _w7 : DINT;
END_VAR

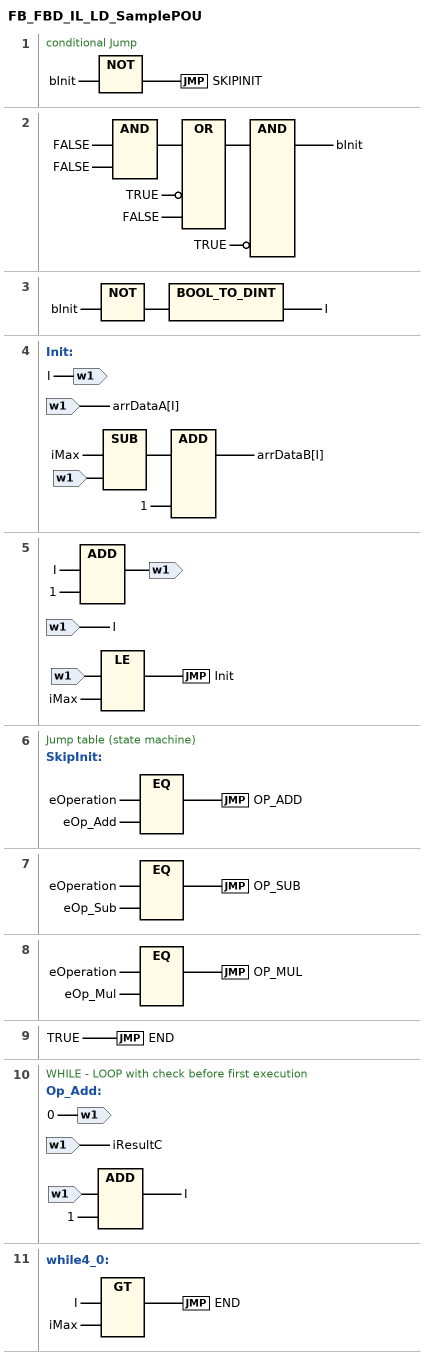
// NETWORK 1
//  conditional Jump
IF NOT bInit THEN JMP SKIPINIT; END_IF

// NETWORK 2
bInit := (FALSE AND FALSE OR NOT TRUE OR FALSE) AND NOT TRUE;

// NETWORK 3
I := BOOL_TO_DINT(NOT bInit);

// NETWORK 4
Init:
arrDataA[I] := I;
arrDataB[I] := (iMax - I) + 1;

// NETWORK 5
_w1 := I + 1;
I := _w1;
IF _w1 <= iMax THEN JMP Init; END_IF

// NETWORK 6
//  Jump table (state machine)
SkipInit:
IF eOperation = eOp_Add THEN JMP OP_ADD; END_IF

// NETWORK 7
IF eOperation = eOp_Sub THEN JMP OP_SUB; END_IF

// NETWORK 8
IF eOperation = eOp_Mul THEN JMP OP_MUL; END_IF

// NETWORK 9
JMP END;

// NETWORK 10
//  WHILE - LOOP with check before first execution
Op_Add:
iResultC := 0;
I := 0 + 1;

// NETWORK 11
while4_0:
IF I > iMax THEN JMP END; END_IF

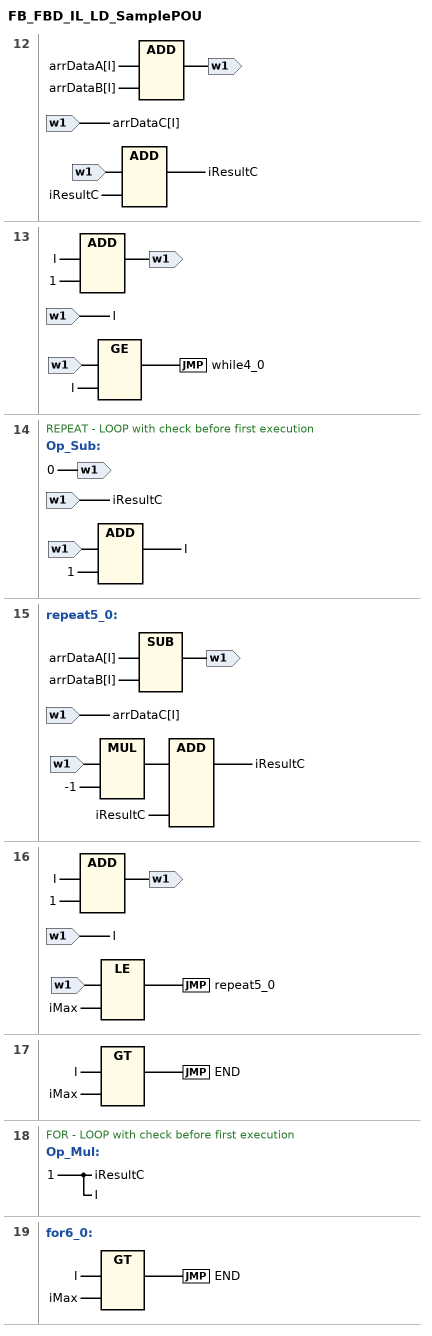
// NETWORK 12
_w2 := arrDataA[I] + arrDataB[I];
arrDataC[I] := _w2;
iResultC := _w2 + iResultC;

// NETWORK 13
_w3 := I + 1;
I := _w3;
IF _w3 >= I THEN JMP while4_0; END_IF

// NETWORK 14
//  REPEAT - LOOP with check before first execution
Op_Sub:
iResultC := 0;
I := 0 + 1;

// NETWORK 15
repeat5_0:
_w4 := arrDataA[I] - arrDataB[I];
arrDataC[I] := _w4;
iResultC := _w4 * -1 + iResultC;

// NETWORK 16
_w5 := I + 1;
I := _w5;
IF _w5 <= iMax THEN JMP repeat5_0; END_IF

// NETWORK 17
IF I > iMax THEN JMP END; END_IF

// NETWORK 18
//  FOR - LOOP with check before first execution
Op_Mul:
iResultC := 1;
I := 1;

// NETWORK 19
for6_0:
IF I > iMax THEN JMP END; END_IF

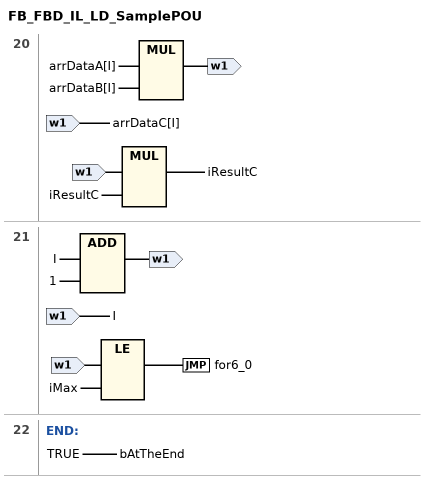
// NETWORK 20
_w6 := arrDataA[I] * arrDataB[I];
arrDataC[I] := _w6;
iResultC := _w6 * iResultC;

// NETWORK 21
_w7 := I + 1;
I := _w7;
IF _w7 <= iMax THEN JMP for6_0; END_IF

// NETWORK 22
END:
bAtTheEnd := TRUE;

END_FUNCTION_BLOCK

// ---- POUs/SampleIEC Languages/MAIN_SFC.TcPOU
PROGRAM MAIN_SFC
VAR
	Timer			: TON;
	fbSFC_SamplePOU : FB_SFC_SamplePou;

	eOperation		: E_Operation := eOp_Add;
	iResultC		: DINT;
	bZero			: BOOL;
	bPos			: BOOL;
	bNeg			: BOOL;
	bTest			: BOOL;
	tTimerValue		: TIME := T#3S;
END_VAR

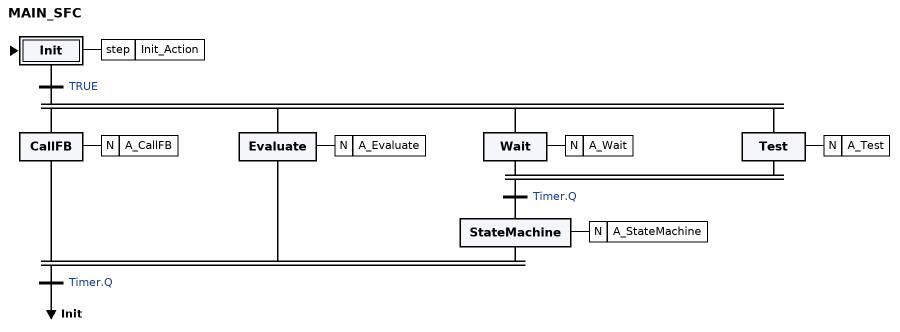
INITIAL_STEP Init:
    Init_Action(N);  // step action
END_STEP
TRANSITION FROM Init TO (CallFB, Evaluate, Wait, Test)
    := TRUE;
END_TRANSITION
STEP CallFB:
    A_CallFB(N);
END_STEP
STEP Evaluate:
    A_Evaluate(N);
END_STEP
STEP Wait:
    A_Wait(N);
END_STEP
STEP Test:
    A_Test(N);
END_STEP
TRANSITION FROM (Wait, Test) TO StateMachine
    := Timer.Q;
END_TRANSITION
STEP StateMachine:
    A_StateMachine(N);
END_STEP
TRANSITION FROM (CallFB, Evaluate, StateMachine) TO Init
    := Timer.Q;
END_TRANSITION

ACTION A_CallFB:
(* FB Call *)
fbSFC_SamplePOU(
	eOperation	:= eOperation,
	iResultC	=> iResultC
);
END_ACTION

ACTION A_Evaluate:
(* Evaluation *)
IF fbSFC_SamplePOU.iResultC = 0 THEN
	bZero := TRUE;
	bPos := FALSE;
	bNeg := FALSE;
ELSIF fbSFC_SamplePOU.iResultC > 0 THEN
	bZero := FALSE;
	bPos := TRUE;
	bNeg := FALSE;
ELSIF fbSFC_SamplePOU.iResultC < 0 THEN
	bZero := FALSE;
	bPos := FALSE;
	bNeg := TRUE;
END_IF
END_ACTION

ACTION A_StateMachine:
(* State machine *)
CASE eOperation OF
eOp_Add:
	eOperation := eOp_MUL;
eOp_Sub:
	eOperation := eOp_ADD;
eOp_Mul:
	eOperation := eOp_SUB;
END_CASE
END_ACTION

ACTION A_Test:
bTest := (((bZero AND bPos) OR (bPos XOR bNeg)) AND (Timer.ET > TIME#500MS) AND (iResultC <= 0)) OR (Timer.ET <= TIME#500MS);
END_ACTION

ACTION A_Wait:
(* Timer *)
Timer(IN := TRUE, PT := tTimerValue);
END_ACTION

ACTION Init_Action:
Timer(IN := FALSE);
END_ACTION

END_PROGRAM

// ---- POUs/SampleIEC Languages/FunctionBlocks/FB_SFC_SamplePou.TcPOU
FUNCTION_BLOCK FB_SFC_SamplePou
VAR_INPUT
//	eOperation	: INT;
	eOperation	: E_Operation;
END_VAR
VAR_OUTPUT
	iResultC	: DINT;
END_VAR
VAR
	arrDataA	: ARRAY [1..iMax] OF DINT;
	arrDataB	: ARRAY [1..iMax] OF DINT;
	arrDataC	: ARRAY [1..iMax] OF DINT;
	I 			: DINT;
	bInit		: BOOL := TRUE;
	bAdd		: BOOL;
	bSub		: BOOL;
	bMul		: BOOL;
END_VAR
VAR CONSTANT
	iMax 		: DINT := 10;
END_VAR

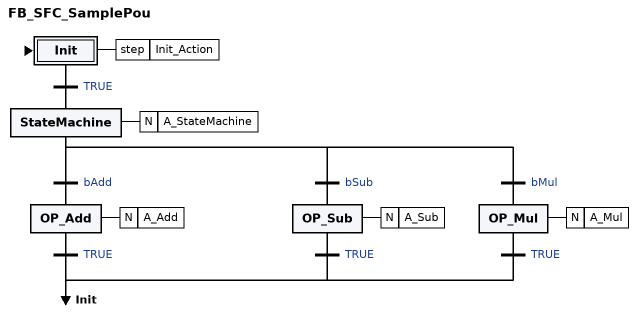
INITIAL_STEP Init:
    Init_Action(N);  // step action
END_STEP
TRANSITION FROM Init TO StateMachine
    := TRUE;
END_TRANSITION
STEP StateMachine:
    A_StateMachine(N);
END_STEP
TRANSITION FROM StateMachine TO OP_Add
    := bAdd;
END_TRANSITION
STEP OP_Add:
    A_Add(N);
END_STEP
TRANSITION FROM OP_Add TO Init
    := TRUE;
END_TRANSITION
TRANSITION FROM StateMachine TO OP_Sub
    := bSub;
END_TRANSITION
STEP OP_Sub:
    A_Sub(N);
END_STEP
TRANSITION FROM OP_Sub TO Init
    := TRUE;
END_TRANSITION
TRANSITION FROM StateMachine TO OP_Mul
    := bMul;
END_TRANSITION
STEP OP_Mul:
    A_Mul(N);
END_STEP
TRANSITION FROM OP_Mul TO Init
    := TRUE;
END_TRANSITION

ACTION A_Add:
(* WHILE - LOOP with check before first execution *)
iResultC := 0;
I := 1;
WHILE I <= iMax DO
	arrDataC[I] := arrDataA[I] + arrDataB[I];
	iResultC 	:= iResultC + arrDataC[I];
	I := I + 1;
END_WHILE
END_ACTION

ACTION A_Mul:
(* FOR - LOOP with check before first execution *)
iResultC := 1;
FOR I := 1 TO iMax DO
	arrDataC[I] := arrDataA[I] * arrDataB[I];
	iResultC 	:= iResultC * arrDataC[I];
END_FOR
END_ACTION

ACTION A_StateMachine:
bAdd := (eOperation = eOp_ADD);
bSub := (eOperation = eOp_SUB);
bMul := (eOperation = eOp_MUL);
END_ACTION

ACTION A_Sub:
(* REPEAT - LOOP: for array access *)
iResultC := 0;
I := 1;
REPEAT
	arrDataC[I] := arrDataA[I] - arrDataB[I];
	iResultC 	:= iResultC - arrDataC[I];
	I := I + 1;
UNTIL I > iMax END_REPEAT
END_ACTION

ACTION Init_Action:
IF bInit THEN
	bInit := FALSE;

	(* FOR loop: for array access *)
	FOR I := 1 TO iMax DO
		arrDataA[I] := I;
		arrDataB[I] := iMax - I + 1;
	END_FOR
END_IF
END_ACTION

END_FUNCTION_BLOCK

// ---- POUs/SampleIEC Languages/MAIN_ST.TcPOU
PROGRAM MAIN_ST
VAR
	Timer			: TON;
	fbST_SamplePOU 	: FB_ST_SamplePOU;

	eOperation		: E_Operation := eOp_Add;
	iResultC		: DINT;
	bZero AT %Q*	: BOOL;
	bPos  AT %Q*	: BOOL;
	bNeg  AT %Q*	: BOOL;
	bTest AT %Q*	: BOOL;
	tTimerValue		: TIME := T#3S;
END_VAR

bTest := (((bZero AND bPos) OR (bPos XOR bNeg)) AND (Timer.ET > TIME#500MS) AND (iResultC <= 0)) OR (Timer.ET <= TIME#500MS);

(* Timer *)
Timer(IN := TRUE, PT := tTimerValue);
IF Timer.Q THEN
	Timer(IN := FALSE);

	(* State machine *)
	CASE eOperation OF
	eOp_Add:
		eOperation := eOp_MUL;
	eOp_Sub:
		eOperation := eOp_ADD;
	eOp_Mul:
		eOperation := eOp_SUB;
	END_CASE
END_IF

(* FB Call *)
fbST_SamplePOU(
	eOperation	:= eOperation,
	iResultC	=> iResultC
);

(* Evaluation *)
IF fbST_SamplePOU.iResultC = 0 THEN
	bZero := TRUE;
	bPos := FALSE;
	bNeg := FALSE;
ELSIF fbST_SamplePOU.iResultC > 0 THEN
	bZero := FALSE;
	bPos := TRUE;
	bNeg := FALSE;
ELSIF fbST_SamplePOU.iResultC < 0 THEN
	bZero := FALSE;
	bPos := FALSE;
	bNeg := TRUE;
END_IF

END_PROGRAM

// ---- POUs/SampleIEC Languages/FunctionBlocks/FB_ST_SamplePOU.TcPOU
FUNCTION_BLOCK FB_ST_SamplePOU
VAR_INPUT
//	eOperation	: INT;
	eOperation	: E_Operation;
END_VAR
VAR_OUTPUT
	iResultC	: DINT;
END_VAR
VAR
	arrDataA	: ARRAY [1..iMax] OF DINT;
	arrDataB	: ARRAY [1..iMax] OF DINT;
	arrDataC	: ARRAY [1..iMax] OF DINT;
	I 			: DINT;
	bInit		: BOOL := TRUE;
END_VAR
VAR CONSTANT
	iMax 		: DINT := 10;
END_VAR

(* IF/ELSE - construct: for conditional code *)
IF bInit THEN
	bInit := FALSE;

	(* FOR loop: for array access *)
	FOR I := 1 TO iMax DO
		arrDataA[I] := I;
		arrDataB[I] := iMax - I + 1;
	END_FOR
END_IF

(* CASE construct: for state machines or switch cases *)
CASE eOperation OF
eOp_Add:
	(* WHILE - LOOP with check before first execution *)
	iResultC := 0;
	I := 1;
	WHILE I <= iMax DO
		arrDataC[I] := arrDataA[I] + arrDataB[I];
		iResultC 	:= iResultC + arrDataC[I];
		I := I + 1;
	END_WHILE

eOp_Sub:
	(* REPEAT - LOOP: for array access *)
	iResultC := 0;
	I := 1;
	REPEAT
		arrDataC[I] := arrDataA[I] - arrDataB[I];
		iResultC 	:= iResultC - arrDataC[I];
		I := I + 1;
	UNTIL I > iMax END_REPEAT

eOp_Mul:
	(* FOR - LOOP with check before first execution *)
	iResultC := 1;
	FOR I := 1 TO iMax DO
		arrDataC[I] := arrDataA[I] * arrDataB[I];
		iResultC 	:= iResultC * arrDataC[I];
	END_FOR
END_CASE

END_FUNCTION_BLOCK

// ---- POUs/IoT and JsonXml/IoT_JSON_XML.TcPOU
PROGRAM IoT_JSON_XML
VAR
	
	//Data Struct and data struct population
	DataValues : IoTDataStruct;
	ReceiveDataValues : IoTDataStruct;
	
	//String send/rec vars
	fb_SendString : FB_MqttCom_String;
	MyRecString: STRING(2000);
	
	//JSON Encoding of Data Struct
	fb_EncodeJSON : FB_JSONEncoding; 
	StringToSend: STRING(2000);
END_VAR

//Populate Data Stuct with data
prgPopulateStructure( DataStructure := DataValues);

//Encode the Data Struct to JSON format
fb_EncodeJSON(DataStruct := DataValues, sJsonDoc2 => StringToSend);

//Send Data Struct as JSON
fb_SendString(sTopicPub:= 'JSON_Data', sPayloadPub:= StringToSend, sTopicSub:= 'JSON_Data', sPayloadRcv => MyRecString);

END_PROGRAM

// ---- POUs/IoT and JsonXml/FBs/FB_MqttCom_String.TcPOU
FUNCTION_BLOCK FB_MqttCom_String
VAR_INPUT
	(* published message *)
	sTopicPub : STRING(255) := 'MyTopic_String';
	sPayloadPub : STRING(255);
	sTopicSub : STRING(255) := 'MyTopic_String';
END_VAR

VAR_OUTPUT
	{attribute 'TcEncoding':='UTF-8'}
	sPayloadRcv : STRING(255);
END_VAR

VAR
	fbMqttClient : FB_IotMqttClient;
	bSetParameter : BOOL := TRUE;
	bConnect : BOOL := TRUE;
	
	
	i: UDINT;
	fbTimer : TON := (PT:=T#1S);
	
	(* received message *)
	bSubscribed : BOOL;
	{attribute 'TcEncoding':='UTF-8'}
	sTopicRcv : STRING(255);

	fbMessageQueue : FB_IotMqttMessageQueue;
	fbMessage : FB_IotMqttMessage;
	
	hrErrorOccurred : HRESULT; // contains the latest occurred error
END_VAR

IF bSetParameter THEN
	bSetParameter := FALSE;
	fbMqttClient.sHostName:= 'localhost';
	fbMqttClient.nHostPort:= 1883;
//	fbMqttClient.sClientId:= 'MyTcMqttClient'; 
	fbMqttClient.sTopicPrefix:= ''; 
	fbMqttClient.ipMessageQueue := fbMessageQueue;
END_IF

fbMqttClient.Execute(bConnect);
IF fbMqttClient.bError THEN
	// add your error logging here
	hrErrorOccurred := fbMqttClient.hrErrorCode;
END_IF

IF fbMessageQueue.nQueuedMessages > 0 THEN
	IF fbMessageQueue.Dequeue(fbMessage:=fbMessage) THEN
		fbMessage.GetTopic(pTopic:=ADR(sTopicRcv), nTopicSize:=SIZEOF(sTopicRcv) );
		fbMessage.GetPayload(pPayload:=ADR(sPayloadRcv), nPayloadSize:=SIZEOF(sPayloadRcv), bSetNullTermination:=FALSE);
	END_IF
END_IF

IF fbMqttClient.bConnected THEN
	IF NOT bSubscribed THEN
		bSubscribed := fbMqttClient.Subscribe(sTopic:=sTopicSub, eQoS:=TcIotMqttQos.AtMostOnceDelivery);
		IF fbMqttClient.bError THEN
			// add your error logging here
			hrErrorOccurred := fbMqttClient.hrErrorCode;
		END_IF
	END_IF
	fbTimer(IN:=TRUE);
	IF fbTimer.Q THEN // publish new payload every second
		fbTimer(IN:=FALSE);
		fbMqttClient.Publish(	sTopic:= sTopicPub, 
								pPayload:= ADR(sPayloadPub), nPayloadSize:= LEN2(ADR(sPayloadPub))+1, 
								eQoS:= TcIotMqttQos.AtMostOnceDelivery, bRetain:= FALSE, bQueue:= FALSE );
		IF fbMqttClient.bError THEN
			// add your error logging here
			hrErrorOccurred := fbMqttClient.hrErrorCode;
		END_IF
	END_IF
END_IF

END_FUNCTION_BLOCK

// ---- POUs/IoT and JsonXml/FBs/FB_JSONEncoding.TcPOU
FUNCTION_BLOCK FB_JSONEncoding
VAR_INPUT
	DataStruct : IoTDataStruct;
END_VAR
VAR_OUTPUT
	sJsonDoc2 : STRING(2000);
END_VAR
VAR
	fbJson : FB_JsonSaxWriter;
	fbJsonDataType : FB_JsonReadWriteDatatype;
	GetTime : FB_LocalSystemTime;
	
	sJsonDoc: STRING(2000);
	
	TimeAsStruct : TIMESTRUCT;

	SystemTime : DATE_AND_TIME;
END_VAR

GetTime(bEnable:= TRUE, dwCycle:=5, systemTime => TimeAsStruct);
SystemTime := SystemTime_to_DT(TimeAsStruct);


fbJson.ResetDocument(); //This method clears current JSON build buffer
fbJson.StartObject(); //Generates new JSON object (inserts open curly bracket)
fbJson.AddKeyDateTime('Timestamp', SystemTime); //Add key called timestamp and insert date
fbJsonDataType.AddJsonKeyValueFromSymbol(fbJson, 'Values', 'ST_Data' , SIZEOF(DataStruct), ADR(DataStruct)); //Adds keys and data based on a structure
fbJsonDataType.AddJsonKeyPropertiesFromSymbol(fbJson, 'MetaData', 'ST_Data', 'Unit|DisplayName');
fbJson.EndObject(); //Ends JSON object (inserts closed curly brace)
sJsonDoc := fbJson.GetDocument();
fbJson.CopyDocument(sJsonDoc2, SIZEOF(sJsonDoc2));

END_FUNCTION_BLOCK

// ---- POUs/IoT and JsonXml/FBs/prgPopulateStructure.TcPOU
PROGRAM prgPopulateStructure
VAR_IN_OUT
	DataStructure : IoTDataStruct;
END_VAR
VAR
	fbGenerateData: FB_GenerateData;	
END_VAR


fbGenerateData();

IF DataStructure.bGenerateData THEN
	DataStructure.Sinus_Slow := fbGenerateData.Sinus_Slow1;
	DataStructure.Puls1 := fbGenerateData.Puls1;
	DataStructure.Puls2 := fbGenerateData.Puls2;
END_IF
IF DataStructure.bClearValues THEN
	DataStructure.Sinus_Slow := 0;
	DataStructure.Puls1 := 0;
	DataStructure.Puls2 := 0;
	DataStructure.bClearValues := FALSE;
END_IF


(*
	strText=> , 
	t=> , 
	Treppe=> , 
	Rampe_Fast=> , 
	Rampe_Slow=> , 
	i=> , 
	Peak=> , 
	GrowSlow=> , 
	iCounter=> , 
	Cosinus_Half=> , 
	Sinus_Fast=> , 
	Sinus_Slow1=> , 
	Sinus_Slow2=> , 
	Sinus_VerySlow=> , 
	Sinus_SqFast=> , 
	Sinus_SqSlow=> , 
	Sinus_Cos_Half=> , 
	SinglePeak=> , 
	phi=> , 
	Ts=> , 
	Rechteck1_1=> , 
	Rechteck2_1=> , 
	Rechteck3_1=> , 
	Puls1=> , 
	Puls2=> , 
	dreieck=> , 
	j=> , 
	k=> , 
	iValue=> , 
	iValueBegin=> , 
	iValueEnd=> , 
	iValueArr=> , 
	iValueArr2=> , 
	bRed=> , 
	bGreen=> , 
	bYellow=> , 
	bBlue=> , 
	bGray=> , 
	bBlue2=> , 
	bGray2=> );
	
	*)

END_PROGRAM

// ---- POUs/Database Server/CSVSample.TcPOU
PROGRAM CSVSample
VAR
	// control of the program
	bStart : BOOL;
	Mode	: E_WriteMode; 
	nState : INT; 
	bError : BOOL := FALSE;
	sError: T_MAXSTRING;

	// fb to control the data communication
	fbCSV_Access: FB_CSV_Access;
	InputData : ST_CSVDataStruct;
	
	// datageneration
	rand: DRAND;
	randomNumber: LREAL;
	fbGetSystemTime: GETSYSTEMTIME;
	fileTime : T_FILETIME;
	
	// repetition
	Count: INT;
	ValuesToWrite: INT := 1000;
	risingTrigger: R_TRIG;
	
	// measure time to execute actions
	Timer : TON;
	t : TIME; 
	
	// destination array of read data
	ReadData: ARRAY[0..4] OF ST_CSVDataStruct;
		
END_VAR

Timer(); 

CASE nState OF 
	
	
	0: // init
 
		Count := 0;
		GenerateData();
		Timer (IN:= FALSE);
		risingTrigger(CLK:= bStart);
		
		IF risingTrigger.Q THEN
			
			bStart := FALSE;
			bError := FALSE;
			sError := '';
			
			Timer (IN:= TRUE, PT := T#1H);
			
			IF mode = E_WriteMode.ePLCDBCmd THEN
				nState := 1;
				
			ELSIF mode = E_WriteMode.ePLCDBWriteStruct THEN
				nState := 11;
				
			ELSIF mode = E_WriteMode.ePLCDBReadStruct THEN
				nState := 21;
				
			END_IF
						
		END_IF
		
	
	1:  // fb_PLCDBCMD
	
		IF fbCSV_Access.Write(2, InputData) THEN
			
			IF fbCSV_Access.bError THEN
				nState := 255;
			ELSE
				Count:= Count+1;
				nState := 2; 
			END_IF	
		
		END_IF

		
	2: // repetitions
		
		IF Count <= ValuesToWrite THEN
			GenerateData(); 
			nState := 1;
		ELSE
			t := Timer.ET;
			nState := 0;
		END_IF
	
	
	11: // fbPLCDBWriteStruct
	
		IF fbCSV_Access.WriteStruct(1, InputData) THEN
			IF fbCSV_Access.bError THEN
				nState := 255;
			ELSE
				Count:= Count+1;
				nState := 12; 
			END_IF		
		END_IF		
		
		
	12: // repetitions
	
		IF Count <= ValuesToWrite THEN
			GenerateData(); 
			nState := 11;
		ELSE
			t := Timer.ET;
			nState := 0;
		END_IF

   
	21:  // fbPLCDBReadStruct
	
		IF fbCSV_Access.ReadStruct(hDBID := 1, pData := ADR(ReadData), cbData := SIZEOF(ReadData)) THEN
			IF fbCSV_Access.bError THEN
				nState := 255;
			ELSE
				nState := 0; 
			END_IF		
		END_IF

	
	255: // error
	
		// request error text
		fbCSV_Access.ipTcResult.RequestEventText(1033, sError, SIZEOF(sError));
		bError := TRUE;

END_CASE

METHOD GenerateData : BOOL
VAR_INPUT
END_VAR

VAR
	
END_VAR
rand(Seed := 1, Num => randomNumber);

InputData.ID := InputData.ID +1; 

InputData.Temperature :=InputData.Temperature  + ((randomNumber-0.5)*10)/5;

rand(Seed := 1, Num => randomNumber);
InputData.Velocity := InputData.Velocity + (randomNumber-0.5);

fbGetSystemTime(timeLoDW => fileTime.dwLowDateTime, timeHiDW => fileTime.dwHighDateTime);
InputData.Timestamp := FILETIME_TO_DT(fileTime);

InputData.Name := 'Water Turbine';
END_METHOD

END_PROGRAM

// ---- POUs/Database Server/FB_CSV_Access.TcPOU
FUNCTION_BLOCK FB_CSV_Access
VAR_INPUT
	
END_VAR
VAR_OUTPUT
	bError : BOOL := FALSE; 
	ipTcResult : I_TcMessage;
END_VAR
VAR

	sCmd : T_MaxString := '{ID};{Timestamp};{Name};{Velocity};{Temperature}'; 
	
	fbPLCDBCmd : FB_PLCDBCmdEvt(sNetID:= '', tTimeout := T#30S);
	
	para : ARRAY [0..4] OF ST_ExpParameter :=[
			(eParaType:= E_ExpParameterType.Int64, nParaSize := 8, sParaName := 'ID'),
			(eParaType:= E_ExpParameterType.DateTime, nParaSize := 4, sParaName := 'Timestamp'),
			(eParaType:= E_ExpParameterType.STRING_, nParaSize := 81, sParaName := 'Name'),
			(eParaType:= E_ExpParameterType.Double64, nParaSize := 8, sParaName := 'Velocity'),
			(eParaType:= E_ExpParameterType.Double64, nParaSize := 8, sParaName := 'Temperature')];

	fbPLCDBWrite: FB_PLCDBWriteEvt(sNetID:= '', tTimeout := T#30S);
	fbPLCDBRead : FB_PLCDBReadEvt(sNetID:= '', tTimeout := T#30S);			
	ColumnNames : ARRAY [0..4] OF STRING(50) := ['ID','Timestamp','Name','Velocity','Temperature'];  

END_VAR

METHOD ReadStruct : BOOL
VAR_INPUT
	hDBID : UDINT;
	
	pData : POINTER TO BYTE; //ARRAY[0..4] OF ST_CSVDataStruct;
	cbData: UDINT;
END_VAR
VAR	
END_VAR
ReadStruct := fbPLCDBRead.ReadStruct(
	hDBID:= hDBID, 
	sTableName:= 'CSV_Sample', 
	pColumnNames:= ADR(ColumnNames), 
	cbColumnNames:= SIZEOF(ColumnNames) , 
	sOrderByColumn:= 'ID', 
	eOrderType := E_OrderType.ASC, 
	nStartIndex:=  0, 
	nRecordCount:= 5, 
	pData:= pData, 
	cbData:= cbData);

IF ReadStruct THEN
	IF fbPLCDBRead.bError THEN
		ipTcResult := fbPLCDBRead.ipTcResult;
		bError:= TRUE;
	END_IF
END_IF
END_METHOD

METHOD Write : BOOL
VAR_INPUT
	hDBID : UDINT;
	InputData: ST_CSVDataStruct;	
END_VAR
Write := fbPLCDBCmd.Execute(
	hDBID:= hDBID, 
	pExpression:= ADR(sCmd), 
	cbExpression:= SIZEOF(sCmd), 
	pData:= ADR(InputData), 
	cbData:= SIZEOF(InputData) , 
	pParameter:=  ADR(para), 
	cbParameter:=SIZEOF(para));
	
IF Write THEN
	IF fbPLCDBCmd.bError THEN
		ipTcResult := fbPLCDBCmd.ipTcResult;
		bError:= TRUE;
	END_IF
END_IF
END_METHOD

METHOD WriteStruct : BOOL
VAR_INPUT
	hDBID : UDINT;
	Data : ST_CSVDataStruct; 
END_VAR
VAR
	
END_VAR
WriteStruct := fbPLCDBWrite.WriteStruct(
	hDBID:= hDBID, 
	sTableName:= 'CSV_Sample', 
	pRecord:= ADR(Data), 
	cbRecord:= SIZEOF(Data), 
	pColumnNames:= ADR(ColumnNames), 
	cbColumnNames:= SIZEOF(ColumnNames) );

IF WriteStruct THEN
	IF fbPLCDBWrite.bError THEN
		ipTcResult := fbPLCDBWrite.ipTcResult;
		bError:= TRUE;
	END_IF
END_IF
END_METHOD

END_FUNCTION_BLOCK

// ---- POUs/MainPOUs/MAINFast.TcPOU
PROGRAM MAINFast
(*******************************************************************************************************
Title				:	Main program fast 
Description			:	Calling the created subroutines (Task 100µs)
Version / Date		:	1.0.0 / 23.05.2016 / created program (Version progress see below)
********************************************************************************************************)
VAR

(* Cycle counter *)
	nCycleCounter							:UDINT;
	
END_VAR
(*******************************************************************************************************
Version / Date / Description:
1.0.0   / 23.05.2016 / created program
********************************************************************************************************)
(* End *)

(* MAIN - 100µs *)

(* THIS CODE IS ONLY AN EXAMPLE - YOU HAVE TO CHECK APTITUDE FOR YOUR APPLICATION *)

(* Cycle counter *)
	nCycleCounter := nCycleCounter + 1;

	IF bMachineSequenzAktiv
	THEN
	
		(* Test Averaging *)
		AverageOut();
		
	END_IF
	
(* End *)

END_PROGRAM

// ---- POUs/XFC/AverageOut.TcPOU
PROGRAM AverageOut
VAR
	
(* Averaging - EL3702 analog input Ch1 oversampling *)
	ni										:UINT;
	fAverageAnalogInputCh1					:REAL;

(* Averaging - EL3702 analog input Ch2 oversampling *)
	fAverageAnalogInputCh2					:REAL;
	aData									:ARRAY[0..99] OF INT;
	nDataArrayCounter						:UINT;

(* Read task target start time *)
	dtActDcTime								:T_DCTIME;
	stActDcTime								:DCTIMESTRUCT;

END_VAR
(* End *)

(* Average out - Cycle Time 100µs - oversampling (Cycle Time 100µs / Factor 10 = 10µs) *)

(* Read task target start time *)
	dtActDcTime := F_GetCurDcTaskTime();
	stActDcTime := DCTIME_TO_DCTIMESTRUCT(dtActDcTime);


(* Averaging - EL3702 analog input Ch1 oversampling *)
	fAverageAnalogInputCh1 := 0.0;
	
	FOR ni := 0 TO 9 BY 1 DO
		fAverageAnalogInputCh1 := fAverageAnalogInputCh1 + INT_TO_REAL(aOsAnalogInR11[ni]);
	END_FOR
	
	fAverageAnalogInputCh1 	  := fAverageAnalogInputCh1 / ni;
	
	nAnalogOutP11 			  := REAL_TO_INT(fAverageAnalogInputCh1);


(* Averaging - EL3702 analog input Ch2 oversampling *)
	fAverageAnalogInputCh2 	  := 0.0;
	
	FOR ni := 0 TO 9 BY 1 DO
		fAverageAnalogInputCh2 	 := fAverageAnalogInputCh2 + INT_TO_REAL(aOsInputFromEL4732Out1[ni]);

		aData[nDataArrayCounter] := aOsInputFromEL4732Out1[ni];
		nDataArrayCounter 	     := nDataArrayCounter + 1;
		
		IF nDataArrayCounter > 99
		THEN
			nDataArrayCounter := 0;
		END_IF
	END_FOR
	
	fAverageAnalogInputCh2 	  := fAverageAnalogInputCh2 / ni;

(* End *)

END_PROGRAM

// ---- POUs/EtherCatDiagnostic/Components/FB_DiagnosticEtherCAT.TcPOU
FUNCTION_BLOCK FB_DiagnosticEtherCAT
VAR_OUTPUT CONSTANT
	
	cMinNumberEcSlaves						:UINT := 0;
	cMaxNumberEcSlaves						:UINT := 100;
	cMinNumberEcFrames						:UINT := 0;
	cMaxNumberEcFrames						:UINT := 9;

END_VAR
VAR_INPUT

	bEnable									:BOOL := FALSE;

END_VAR
VAR_OUTPUT

	nFrmXWcState 					AT%I*	:ARRAY[cMinNumberEcFrames..cMaxNumberEcFrames] OF UINT;
	nDevState 						AT%I*	:UINT;
	sDevState								:STRING;
	nDevId 							AT%I*	:UINT;
	cbAmsNetId 						AT%I*	:ARRAY[0..5] OF BYTE;
	sNetIdText 								:STRING;
	nCfgSlaveCount					AT%I*	:UINT;
	
(* Evaluated terminal diagnose info *)
	stEcTerminalDiagInfo 					:ARRAY[cMinNumberEcSlaves..cMaxNumberEcSlaves] OF ST_EcTerminalDiagInfo;

(* Read configured EtherCAT System *)
	bEcSystemRead							:BOOL;

END_VAR
VAR
{attribute 'hide'}
(* Read configured EtherCAT System *)
	bStartDiag								:BOOL;
	eStatus1								:E_EcSystemStatus;
	fbEcGetConfSlaves 						:FB_EcGetConfSlaves;
	stEcConfigSlaveData						:ARRAY[cMinNumberEcSlaves..cMaxNumberEcSlaves] OF ST_EcSlaveConfigData;
	nNumberConfEcMember						:UINT;

(* Read EtherCAT diagnosis and change the master status state*)
	eStatus2								:E_EcDiacStatus;
	nAltFrmXWcState							:ARRAY[cMinNumberEcFrames..cMaxNumberEcFrames] OF UINT;
	nAltDevState							:UINT;
	fbEcGetMasterState						:FB_EcGetMasterState;
	nStatusMaster							:WORD;
	sMasterText								:STRING;

	stSlaveStatus							:ARRAY[cMinNumberEcSlaves..cMaxNumberEcSlaves] OF ST_EcSlaveState;
	sDeviceStatusText						:ARRAY[cMinNumberEcSlaves..cMaxNumberEcSlaves] OF STRING;
	ni										:UINT;
	fbTon									:TON;
	fbEcGetAllSlaveStates					:FB_EcGetAllSlaveStates;

END_VAR
(* End *)

(* diagnosis of the EtherCat System *)

(* Create the NetId-String *)
	sNetIdText := F_CreateAmsNetId(cbAmsNetId);

(* Create the DevState-String *)	
	sDevState := F_ConvMasterDevStateToString(nDevState);

(* Read configured EtherCAT System *)
	act_RdEcSystem();

(* Read EtherCAT master and slave diagnosis states *)
	act_RwEcDiagnose();
	
(* End *)

ACTION act_RdEcSystem:
(* Read configured EtherCAT System *)

	CASE eStatus1 OF

		eEcSystem_Start				:	(* Start reading *)

			IF bEnable 
				AND NOT bEcSystemRead
				AND sNetIdText <> '0.0.0.0.0.0'
			THEN
				eStatus1 := eEcSystem_ReadConfSystem;
			END_IF

		eEcSystem_ReadConfSystem	:	(* Read configured EtherCAT System *)

			fbEcGetConfSlaves(	
				sNetId				:= 	sNetIdText,
				pArrEcConfSlaveInfo	:= 	ADR(stEcConfigSlaveData),
				cbBufLen			:= 	SIZEOF(stEcConfigSlaveData),
				bExecute			:= 	TRUE,
				tTimeout			:= 	DEFAULT_ADS_TIMEOUT,
				nSlaves				=> 	nNumberConfEcMember);

			IF NOT fbEcGetConfSlaves.bBusy
				AND NOT fbEcGetConfSlaves.bError
			THEN

				FOR ni := cMinNumberEcSlaves TO cMaxNumberEcSlaves BY 1 DO
					stEcTerminalDiagInfo[ni].nAddr := stEcConfigSlaveData[ni].nAddr;
					stEcTerminalDiagInfo[ni].sType := stEcConfigSlaveData[ni].sType;
					stEcTerminalDiagInfo[ni].sName := stEcConfigSlaveData[ni].sName;
				END_FOR

				fbEcGetConfSlaves(bExecute := FALSE);
				bEcSystemRead 	:= TRUE;
				bStartDiag 		:= TRUE;
				eStatus1   		:= eEcSystem_Start;

			END_IF

	END_CASE

(* End *)
END_ACTION

ACTION act_RwEcDiagnose:
(* Read EtherCAT master and slave diagnosis states *)

	CASE eStatus2 OF

		eEcDiac_Start				:	(* Start reading *)

			(* Check master device state of first diag run *)
			IF (nDevState <> nAltDevState)
				OR bStartDiag
			THEN 
				bStartDiag 			:= FALSE;
				nAltDevState 		:= nDevState;
				eStatus2   			:= eEcDiac_Delay;
			END_IF
			
			(* Check frame status *)
			FOR ni := cMinNumberEcFrames TO cMaxNumberEcFrames BY 1 DO
				IF nFrmXWcState[ni] <> nAltFrmXWcState[ni]
				THEN	
					eStatus2   			:= eEcDiac_Delay;
				END_IF
				nAltFrmXWcState[ni]	:= nFrmXWcState[ni];
			END_FOR
			
		eEcDiac_Delay				:	(* Delay - read diagnosis *)

				fbTon(	IN	:=	TRUE,
						PT	:=	t#400ms);

				IF fbTon.Q
				THEN
					fbTon(IN := FALSE);
					eStatus2 := eEcDiac_ReadMasterState;
				END_IF


		eEcDiac_ReadMasterState		:	(* Read master state *)

				fbEcGetMasterState(	
					sNetId		:=	sNetIdText,
					bExecute	:=	TRUE,
					tTimeout	:=	T#1s,
					bBusy		=> 	,
					bError		=> 	,
					nErrId		=> 	,
					state		=>	nStatusMaster);

				IF NOT fbEcGetMasterState.bBusy
				THEN

					fbEcGetMasterState(bExecute := FALSE);
					eStatus2 := eEcDiac_ReadSlaveState;

					sMasterText := F_ConvStateToString(nStatusMaster);
				END_IF


		eEcDiac_ReadSlaveState		:	(* Read all slave states *)

				fbEcGetAllSlaveStates(	
					sNetId		:=	sNetIdText,
					pStateBuf	:=	ADR(stSlaveStatus),
					cbBufLen	:=	SIZEOF(stSlaveStatus),
					bExecute	:=	TRUE,
					tTimeout	:=	t#1s);

				IF NOT fbEcGetAllSlaveStates.bBusy
				THEN

					fbEcGetAllSlaveStates(bExecute := FALSE);

					FOR ni := cMinNumberEcSlaves TO cMaxNumberEcSlaves BY 1 DO

						sDeviceStatusText[ni] := F_ConvSlaveStateToString(stSlaveStatus[ni]);
						stEcTerminalDiagInfo[ni].sTerminalStatus := sDeviceStatusText[ni];

					END_FOR

					eStatus2 := eEcDiac_Start;

				END_IF

	END_CASE

(* End *)
END_ACTION

END_FUNCTION_BLOCK

// ---- POUs/RT Monitor/simpleMarksPrg.TcPOU
PROGRAM simpleMarksPrg
VAR
	// Instance of the function block for using the "simple" marks
	
	fblog : fb_RTmon_LogMark;
END_VAR

fblog.LogStart(100,0);


// process counting, sequence start
IF GVL.fbCrititcalSection.Enter() THEN
	GVL.iGlobalCounter:=GVL.iGlobalCounter+1;
	ConsumeTime(50);
    GVL.fbCrititcalSection.Leave();
END_IF

fblog.LogStop(100,0);

END_PROGRAM

// ---- POUs/TwinSAFE/Components/FB_TwinSafeConnectionEK1914.TcPOU
FUNCTION_BLOCK FB_TwinSafeConnectionEK1914
(*******************************************************************************************************
Description			:	Evaluate a TwinSAFE connection status and diagnosis to an EtherCAT terminal
Supported terminals : 	EK1914
Documentation 		:	EK1914 TwinSAFE input/output terminal with 2 fail-safe inputs and 2 fail-safe outputs
Version/Date 		:	V1.2.0/08.03.2016
Required libraries 	: 	TcSystem.lib (Tc2_System), TcEtherCAT.lib (Tc2_EtherCAT)
********************************************************************************************************)
VAR_INPUT
	
	tCoEReadCycle							:TIME 	:= T#0MS;				(* Read cycle CoE-Data, e.g. temperature *)

END_VAR
VAR_OUTPUT

	stInfoData						AT %I*	:ST_TsConnectionInfo2Byte;		(* EL6900 \ Connection Info Data \ Message_X Info Data*)
	nEcSlaveState					AT %I*	:UINT ;							(* EK1914 \ InfoData \ State *)
	stEcAdsAddr						AT %I*	:ST_AdsAddr;					(* EK1914 \ InfoData \ AdsAddr *)

(* act_EcSlaveIdentify *)
	sEcSlaveType							:STRING(15);
	sEcSlaveName							:STRING(31) := '';
	bSlaveIdentify							:BOOL;
	bSlaveTypeError							:BOOL;
	
(* act_Signals *)
	bChannel1In								:BOOL;							
	bChannel2In								:BOOL;
	bChannel1Out							:BOOL;
	bChannel2Out							:BOOL;

(* act_ConnectionState *)
	sState									:STRING;
	
(* act_ConnectionDiag *)
	sDiag									:STRING;
	sFault									:STRING;						(* FailSafe Error (Hardware)*)
	bError									:BOOL;							(* TwinSAFE-Error *)
	
(* act_ReadDiagObjects *)
	stSlaveTemp								:ST_TsSlave2Temp;
	bTempWarning							:BOOL;							(* Temperature warning: T1, T2, TOut *)
	stTsDiagObjectsBitsEK1914				:ST_TsDiagObjectsBitsEK1914;

END_VAR
VAR

(* act_ConnectionDiag *)
	nDiag0_3								:BYTE;

(* act_ReadDiagObjects *)
	eReadDiagObjState						:E_TsCycleDiagObj;
	eReadDiagObjErrStep						:E_TsCycleDiagObj := E_TsCycleDiagObj.eCycleDiagObj_NoError;
	bReadDiagObjError						:BOOL;							(* Error in the diagnosis objects read cycle *)  
	bReadDiagObjReset						:BOOL;							(* Reset the diagnosis objects read cycle error *)
	fbTimer									:TON;
	fbEcCoeSdoRead							:FB_EcCoESdoReadEx;
	fbEcCoeSdoReadT2						:FB_EcCoESdoReadEx;
	stDiagObjects							:ST_TsDiagObjectsEK1914;

(* act_EcSlaveIdentify *)
	fbEcGetSlaveName						:FB_EcGetSlaveName;

END_VAR
VAR CONSTANT
	
(* act_ReadDiagObjects *)
	nWarningLevelTemp1						:INT	:= 85;					(* Temperature 1 warning level [°C] *)
	nWarningLevelTemp2						:INT	:= 85;					(* Temperature 2 warning level [°C] *)

END_VAR
(* End *)

(* Function Block TwinSAFE connection status and diagnosis for EL1904 Terminals *)

(* THIS CODE IS ONLY AN EXAMPLE - YOU HAVE TO CHECK APTITUDE FOR YOUR APPLICATION *)

	(* Identify the EtherCAT slave *)
		act_EcSlaveIdentify();

	(* Evaluate the connection state *)
		act_ConnectionState();
	
	(* Evaluate the connection diagnosis *)
		act_ConnectionDiag();
	
	(* Evaluate the EL1904 input signals *)
		act_Signals();
	
	(* Evaluate the Terminal temperatures and diagnostic objects *)
		IF bSlaveIdentify
		THEN
			act_ReadDiagObjects();
		ELSE
			eReadDiagObjState := E_TsCycleDiagObj.eCycleDiagObj_Init;
		END_IF

	
(* End *)

ACTION act_ConnectionDiag:
(* Evaluate the connection diagnosis *)

	(* Evaluate Bit 0..3 *)
	nDiag0_3 := USINT_TO_BYTE(stInfoData.nDiag) AND 16#0F;

	CASE nDiag0_3 OF
		0:		sDiag := 'No error';
		1:		sDiag := 'Invalid command';
		2:		sDiag := 'Unknown command';
		3:		sDiag := 'Invalid connection ID';
		4:		sDiag := 'Invalid CRC';
		5:		sDiag := 'Watchdog time elapsed';
		6:		sDiag := 'Invalid FSOE address';
		7:		sDiag := 'Invalid data';
		8:		sDiag := 'Invalid communication parameter length';
		9:		sDiag := 'Invalid communication parameters';
		10:		sDiag := 'Invalid user parameter length';
		11:		sDiag := 'Invalid user parameter';
		12:		sDiag := 'FSoE master reset';
		13:		sDiag := 'Module err detected on slave, with option "Module error is ComError" activated';
		14:		sDiag := 'Module err detected on EL290x, with option "Error acknowledge active" activated';
		15:		sDiag := 'Slave not yet started, or unexpected error argument';
	END_CASE

	(* Evaluate Bit 4..7 *)
	sFault:='';

	IF stInfoData.nDiag.4 
	THEN
		sFault	:= 'FSoE slave error detected - '; 
	END_IF

	IF stInfoData.nDiag.5 
	THEN
		sFault	:= concat(sFault,'FSoE slave reports Failsafe Value active - ');
	END_IF

	IF stInfoData.nDiag.6 
	THEN
		sFault	:= concat(sFault,'StartUp - ');
	END_IF

	IF stInfoData.nDiag.7 
	THEN
		sFault	:= concat(sFault, 'FSoE master reports Failsafe Value active');
	END_IF
		
	(* Error *)
	bError := stInfoData.nDiag <> 0;

(* End *)
END_ACTION

ACTION act_ConnectionState:
(* Evaluate the connection state *)

	CASE stInfoData.nState OF
		100:	sState := 'Reset state';
		101:	sState := 'Session state';
		102:	sState := 'Connection state';
		103:	sState := 'Parameter state';
		104:	sState := 'Data state';
		105:	sState := 'Shutdown state';
	ELSE
		sState := 'unknown';
	END_CASE
	
(* End *)
END_ACTION

ACTION act_DiagObjectsBits:
(* act_TsDiagObjectsBits *)

	stTsDiagObjectsBitsEK1914.bErrInput1		 			:= stDiagObjects.nSensorTestError.0;
	stTsDiagObjectsBitsEK1914.bErrInput2		 			:= stDiagObjects.nSensorTestError.1;

	stTsDiagObjectsBitsEK1914.bErrFirstInputPair		 	:= stDiagObjects.nDuringTwoChannelEvaluationError.0;

	stTsDiagObjectsBitsEK1914.bMatOpModeErrFirstInputPair	:= stDiagObjects.nMatModeInputPairDisagreeError.0
																	AND stDiagObjects.nMatModeInputPairDisagreeError.1;
	
	stTsDiagObjectsBitsEK1914.bMatOpModeExtSupplyErrInput1	:= stDiagObjects.nMatModeExternalSupplyError.0;
	stTsDiagObjectsBitsEK1914.bMatOpModeExtSupplyErrInput2	:= stDiagObjects.nMatModeExternalSupplyError.1;

	stTsDiagObjectsBitsEK1914.bCcErrOutput1	 				:= stDiagObjects.nDiagnosisMicroC1 = 5;
	stTsDiagObjectsBitsEK1914.bCcErrOutput2	 				:= stDiagObjects.nDiagnosisMicroC1 = 6;
	stTsDiagObjectsBitsEK1914.bOvervoltage	 				:= stDiagObjects.nDiagnosisMicroC1 = 10;
	stTsDiagObjectsBitsEK1914.bUndervoltage	 				:= stDiagObjects.nDiagnosisMicroC1 = 11;
	stTsDiagObjectsBitsEK1914.bErrTestFieldVolSitches	 	:= stDiagObjects.nDiagnosisMicroC1 >= 21
																	AND stDiagObjects.nDiagnosisMicroC1 <= 27;
	stTsDiagObjectsBitsEK1914.bErrStartUpOutputCircuit	 	:= stDiagObjects.nDiagnosisMicroC1 >= 30
																	AND stDiagObjects.nDiagnosisMicroC1 <= 33;
	stTsDiagObjectsBitsEK1914.bExtSupply0VOutput1MicroC1	:= stDiagObjects.nDiagnosisMicroC1 = 101;
	stTsDiagObjectsBitsEK1914.bExtSupply24VOutput1MicroC1	:= stDiagObjects.nDiagnosisMicroC1 = 102;
	stTsDiagObjectsBitsEK1914.bExtSupply0VOutput2MicroC1	:= stDiagObjects.nDiagnosisMicroC1 = 103;
	stTsDiagObjectsBitsEK1914.bExtSupply24VOutput2MicroC1	:= stDiagObjects.nDiagnosisMicroC1 = 104;

	stTsDiagObjectsBitsEK1914.bExtSupply0VOutput1MicroC2	:= stDiagObjects.nDiagnosisMicroC2 = 201;
	stTsDiagObjectsBitsEK1914.bExtSupply24VOutput1MicroC2	:= stDiagObjects.nDiagnosisMicroC2 = 202;
	stTsDiagObjectsBitsEK1914.bExtSupply0VOutput2MicroC2	:= stDiagObjects.nDiagnosisMicroC2 = 203;
	stTsDiagObjectsBitsEK1914.bExtSupply24VOutput2MicroC2	:= stDiagObjects.nDiagnosisMicroC2 = 204;
	
(* End *)
END_ACTION

ACTION act_EcSlaveIdentify:
(* Identify the EtherCAT slave *)

	IF NOT nEcSlaveState.3
	THEN
		bSlaveIdentify  := FALSE;
		bSlaveTypeError := FALSE;
		sEcSlaveType    := '';
	END_IF

	IF nEcSlaveState.3
		AND NOT bSlaveIdentify
		AND NOT bSlaveTypeError
 		AND F_CreateAmsNetId(stEcAdsAddr.netId) <> '0.0.0.0.0.0' 
		AND stEcAdsAddr.port <> 0
	THEN

		fbEcCoeSdoRead(
			sNetId			:= 	F_CreateAmsNetId(stEcAdsAddr.netId),
			nSlaveAddr		:= 	stEcAdsAddr.port,
			nSubIndex		:= 	0,
			nIndex			:= 	16#1008,
			pDstBuf			:= 	ADR(sEcSlaveType),
			cbBufLen		:= 	SIZEOF(sEcSlaveType),
			bExecute		:= 	TRUE,
			tTimeout		:= 	DEFAULT_ADS_TIMEOUT);
	

		fbEcGetSlaveName(
			bExecute		:=	TRUE, 
			sNetId			:=	F_CreateAmsNetId(stEcAdsAddr.netId), 
			nSlaveAddr		:=	stEcAdsAddr.port, 
			tTimeout		:=	DEFAULT_ADS_TIMEOUT, 
			bBusy			=>	, 
			sSlaveName		=>	sEcSlaveName, 
			bError			=>	, 
			nErrId			=>	);

		IF NOT fbEcCoeSdoRead.bBusy
			AND NOT fbEcCoeSdoRead.bError
			AND NOT fbEcGetSlaveName.bBusy
			AND NOT fbEcGetSlaveName.bError
		THEN
		
			fbEcCoeSdoRead(bExecute := FALSE); 
			fbEcGetSlaveName(bExecute := FALSE); 

			IF sEcSlaveType = 'EK1914' 
				AND fbEcGetSlaveName.sSlaveName <> ''
			THEN
				bSlaveIdentify := TRUE;
			ELSE
				bSlaveTypeError := TRUE;
			END_IF

		ELSIF NOT fbEcCoeSdoRead.bBusy
			AND fbEcCoeSdoRead.bError
		OR (NOT fbEcGetSlaveName.bBusy
			AND fbEcGetSlaveName.bError)
		THEN
		
			fbEcCoeSdoRead(bExecute := FALSE); 
			fbEcGetSlaveName(bExecute := FALSE); 

		END_IF

	END_IF
	
(* End *)
END_ACTION

ACTION act_ReadDiagObjects:
(* Evaluate the Terminal temperatures and diagnostic objects *)

	CASE eReadDiagObjState OF

		eCycleDiagObj_Init				:	(* Init *)	

			IF nEcSlaveState.3					(* Slave in OP *)
				AND tCoEReadCycle <> T#0MS 		(* tCoEReadCycle <> t#0ms -> Read diagnostic aktiv *)
			THEN
				bReadDiagObjError := FALSE;
				fbEcCoeSdoRead(bExecute := FALSE);
				fbEcCoeSdoReadT2(bExecute := FALSE);
				fbTimer(IN := FALSE);
				eReadDiagObjState := eCycleDiagObj_ReadTemperature;
			END_IF

			
		eCycleDiagObj_ReadTemperature	:	(* Read temperature *)

			fbEcCoeSdoRead(
				sNetId			:= 	F_CreateAmsNetId(stEcAdsAddr.netId),
				nSlaveAddr		:= 	stEcAdsAddr.port,
				nSubIndex		:= 	1,
				nIndex			:= 	16#FA80,
				pDstBuf			:= 	ADR(stSlaveTemp.nInternalTemperature1),
				cbBufLen		:= 	2,
				bExecute		:= 	TRUE,
				tTimeout		:= 	DEFAULT_ADS_TIMEOUT,
				bCompleteAccess	:= 	FALSE);

			fbEcCoeSdoReadT2(
				sNetId			:= 	F_CreateAmsNetId(stEcAdsAddr.netId),
				nSlaveAddr		:= 	stEcAdsAddr.port,
				nSubIndex		:= 	2,
				nIndex			:= 	16#FA80,
				pDstBuf			:= 	ADR(stSlaveTemp.nInternalTemperature2),
				cbBufLen		:= 	2,
				bExecute		:= 	TRUE,
				tTimeout		:= 	DEFAULT_ADS_TIMEOUT,
				bCompleteAccess	:= 	FALSE);

			IF NOT fbEcCoeSdoRead.bBusy 
				AND NOT fbEcCoeSdoRead.bError 
			AND NOT fbEcCoeSdoReadT2.bBusy 
				AND NOT fbEcCoeSdoReadT2.bError 
			THEN
				fbEcCoeSdoRead(bExecute   := FALSE);
				fbEcCoeSdoReadT2(bExecute := FALSE);
				eReadDiagObjState := eCycleDiagObj_ReadDelay;
////			eReadDiagObjState := eCycleDiagObj_ReadDiag;
			ELSIF (NOT fbEcCoeSdoRead.bBusy 
				AND fbEcCoeSdoRead.bError)
 				OR (NOT fbEcCoeSdoRead.bBusy 
				AND fbEcCoeSdoRead.bError) 
			THEN
				eReadDiagObjErrStep := eReadDiagObjState;
				eReadDiagObjState 	:= eCycleDiagObj_Error;
			END_IF

			
		eCycleDiagObj_ReadDiag			:	(* Read diacnostic objects *)

			fbTimer(IN := TRUE, PT := tCoEReadCycle);

			fbEcCoeSdoRead(
				sNetId			:= 	F_CreateAmsNetId(stEcAdsAddr.netId),
				nSlaveAddr		:= 	stEcAdsAddr.port,
				nSubIndex		:= 	1,
				nIndex			:= 	16#800E,
				pDstBuf			:= 	ADR(stDiagObjects),
				cbBufLen		:= 	SIZEOF(stDiagObjects),
				bExecute		:= 	TRUE,
				tTimeout		:= 	DEFAULT_ADS_TIMEOUT,
				bCompleteAccess	:= 	TRUE);

			IF NOT fbEcCoeSdoRead.bBusy 
				AND NOT fbEcCoeSdoRead.bError 
			THEN
				fbEcCoeSdoRead(bExecute := FALSE);
				act_DiagObjectsBits();
				eReadDiagObjState := eCycleDiagObj_ReadDelay;
			ELSIF NOT fbEcCoeSdoRead.bBusy 
				AND fbEcCoeSdoRead.bError 
			THEN
				eReadDiagObjErrStep := eReadDiagObjState;
				eReadDiagObjState 	:= eCycleDiagObj_Error;
			END_IF
				
			
		eCycleDiagObj_ReadDelay		:	(* Read delay *)
			fbTimer(
				IN := TRUE, 
				PT := tCoEReadCycle);

			IF fbTimer.Q 
			THEN
				fbTimer(IN := FALSE); 			
				eReadDiagObjState := eCycleDiagObj_Done;
			END_IF

			
		eCycleDiagObj_Done				:	(* Done *)

			eReadDiagObjState := eCycleDiagObj_Init;

			
		eCycleDiagObj_Error			:	(* Error detected *)

			bReadDiagObjError := TRUE;
		
			IF bReadDiagObjReset
			THEN
				bReadDiagObjError := FALSE;
				fbEcCoeSdoRead(bExecute := FALSE);
				fbEcCoeSdoReadT2(bExecute := FALSE);
				eReadDiagObjErrStep := E_TsCycleDiagObj.eCycleDiagObj_NoError;
				eReadDiagObjState := eCycleDiagObj_Init;
			END_IF

	ELSE
		
		eReadDiagObjState := eCycleDiagObj_Init;
		
	END_CASE

	bTempWarning := stSlaveTemp.nInternalTemperature1 >= nWarningLevelTemp1 
						OR stSlaveTemp.nInternalTemperature2 >= nWarningLevelTemp2;

(* End *)
END_ACTION

ACTION act_Signals:
(* Evaluate the input and output signals *)

	IF nEcSlaveState.3 (* Slave in operational state *)
	THEN
		(* OP -> transfer the signal states *)
		bChannel1In  := stInfoData.nInOutSafeDataByte1.0;
		bChannel2In  := stInfoData.nInOutSafeDataByte1.1;
		bChannel1Out := stInfoData.nInOutSafeDataByte2.0;
		bChannel2Out := stInfoData.nInOutSafeDataByte2.1;
	ELSE
		(* Error -> clear the signal states *)
		bChannel1In := bChannel2In := bChannel1Out := bChannel2Out := FALSE;
	END_IF

(* End *)
END_ACTION

END_FUNCTION_BLOCK

// ---- POUs/TwinSAFE/Components/FB_TwinSafeConnectionEL3214.TcPOU
FUNCTION_BLOCK FB_TwinSafeConnectionEL3214
(*******************************************************************************************************
Description			:	Evaluate a TwinSAFE connection status and diagnosis to an EtherCAT terminal
Supported terminals : 	EL3214-0090
Documentation 		:	
Version/Date 		:	
Required libraries 	: 	TcSystem.lib (Tc2_System), TcEtherCAT.lib (Tc2_EtherCAT)
********************************************************************************************************)
VAR_INPUT
END_VAR
VAR_OUTPUT

	stInfoData						AT %I*	:ST_TsConnectionInfoEL3214;		(* EL6900 \ Connection Info Data \ Message_X Info Data*)
	nEcSlaveState					AT %I*	:UINT ;							(* EL3214-0090 \ InfoData \ State *)
	stEcAdsAddr						AT %I*	:ST_AdsAddr;					(* EL3214-0090 \ InfoData \ AdsAddr *)

(* act_EcSlaveIdentify *)
	sEcSlaveType							:STRING(15);
	sEcSlaveName							:STRING(31) := '';
	bSlaveIdentify							:BOOL;
	bSlaveTypeError							:BOOL;
	
(* act_Signals *)
	nInSafeDataValue1						:UINT;
	nInSafeDataValue2						:INT;
	nInSafeDataValue3						:INT;
	nInSafeDataValue4						:INT;

(* act_ConnectionState *)
	sState									:STRING;
	
(* act_ConnectionDiag *)
	sDiag									:STRING;
	sFault									:STRING;						(* FailSafe Error (Hardware)*)
	bError									:BOOL;							(* TwinSAFE-Error *)
	
END_VAR
VAR

(* act_ConnectionDiag *)
	nDiag0_3								:BYTE;

(* act_EcSlaveIdentify *)
	fbEcCoeSdoRead							:FB_EcCoESdoReadEx;
	fbEcGetSlaveName						:FB_EcGetSlaveName;

END_VAR
(* End *)

(* Function Block TwinSAFE connection status and diagnosis for EL1904 Terminals *)

(* THIS CODE IS ONLY AN EXAMPLE - YOU HAVE TO CHECK APTITUDE FOR YOUR APPLICATION *)

	(* Identify the EtherCAT slave *)
		act_EcSlaveIdentify();

	(* Evaluate the connection state *)
		act_ConnectionState();
	
	(* Evaluate the connection diagnosis *)
		act_ConnectionDiag();
	
	(* Evaluate the EL3214 input signals *)
		act_Signals();
	
(* End *)

ACTION act_ConnectionDiag:
(* Evaluate the connection diagnosis *)

	(* Evaluate Bit 0..3 *)
	nDiag0_3 := USINT_TO_BYTE(stInfoData.nDiag) AND 16#0F;

	CASE nDiag0_3 OF
		0:		sDiag := 'No error';
		1:		sDiag := 'Invalid command';
		2:		sDiag := 'Unknown command';
		3:		sDiag := 'Invalid connection ID';
		4:		sDiag := 'Invalid CRC';
		5:		sDiag := 'Watchdog time elapsed';
		6:		sDiag := 'Invalid FSOE address';
		7:		sDiag := 'Invalid data';
		8:		sDiag := 'Invalid communication parameter length';
		9:		sDiag := 'Invalid communication parameters';
		10:		sDiag := 'Invalid user parameter length';
		11:		sDiag := 'Invalid user parameter';
		12:		sDiag := 'FSoE master reset';
		13:		sDiag := 'Module err detected on slave, with option "Module error is ComError" activated';
		14:		sDiag := 'Module err detected on EL290x, with option "Error acknowledge active" activated';
		15:		sDiag := 'Slave not yet started, or unexpected error argument';
	END_CASE

	(* Evaluate Bit 4..7 *)
	sFault:='';

	IF stInfoData.nDiag.4 
	THEN
		sFault	:= 'FSoE slave error detected - '; 
	END_IF

	IF stInfoData.nDiag.5 
	THEN
		sFault	:= concat(sFault,'FSoE slave reports Failsafe Value active - ');
	END_IF

	IF stInfoData.nDiag.6 
	THEN
		sFault	:= concat(sFault,'StartUp - ');
	END_IF

	IF stInfoData.nDiag.7 
	THEN
		sFault	:= concat(sFault, 'FSoE master reports Failsafe Value active');
	END_IF
		
	(* Error *)
	bError := stInfoData.nDiag <> 0;

(* End *)
END_ACTION

ACTION act_ConnectionState:
(* Evaluate the connection state *)

	CASE stInfoData.nState OF
		100:	sState := 'Reset state';
		101:	sState := 'Session state';
		102:	sState := 'Connection state';
		103:	sState := 'Parameter state';
		104:	sState := 'Data state';
		105:	sState := 'Shutdown state';
	ELSE
		sState := 'unknown';
	END_CASE
	
(* End *)
END_ACTION

ACTION act_EcSlaveIdentify:
(* Identify the EtherCAT slave *)

	IF NOT nEcSlaveState.3
	THEN
		bSlaveIdentify  := FALSE;
		bSlaveTypeError := FALSE;
		sEcSlaveType    := '';
	END_IF

	IF nEcSlaveState.3
		AND NOT bSlaveIdentify
		AND NOT bSlaveTypeError
 		AND F_CreateAmsNetId(stEcAdsAddr.netId) <> '0.0.0.0.0.0' 
		AND stEcAdsAddr.port <> 0
	THEN

		fbEcCoeSdoRead(
			sNetId			:= 	F_CreateAmsNetId(stEcAdsAddr.netId),
			nSlaveAddr		:= 	stEcAdsAddr.port,
			nSubIndex		:= 	0,
			nIndex			:= 	16#1008,
			pDstBuf			:= 	ADR(sEcSlaveType),
			cbBufLen		:= 	SIZEOF(sEcSlaveType),
			bExecute		:= 	TRUE,
			tTimeout		:= 	DEFAULT_ADS_TIMEOUT);
	

		fbEcGetSlaveName(
			bExecute		:=	TRUE, 
			sNetId			:=	F_CreateAmsNetId(stEcAdsAddr.netId), 
			nSlaveAddr		:=	stEcAdsAddr.port, 
			tTimeout		:=	DEFAULT_ADS_TIMEOUT, 
			bBusy			=>	, 
			sSlaveName		=>	sEcSlaveName, 
			bError			=>	, 
			nErrId			=>	);

		IF NOT fbEcCoeSdoRead.bBusy
			AND NOT fbEcCoeSdoRead.bError
			AND NOT fbEcGetSlaveName.bBusy
			AND NOT fbEcGetSlaveName.bError
		THEN
		
			fbEcCoeSdoRead(bExecute := FALSE); 
			fbEcGetSlaveName(bExecute := FALSE); 

			IF sEcSlaveType = 'EL3214-0090' 
				AND fbEcGetSlaveName.sSlaveName <> ''
			THEN
				bSlaveIdentify := TRUE;
			ELSE
				bSlaveTypeError := TRUE;
			END_IF

		ELSIF NOT fbEcCoeSdoRead.bBusy
			AND fbEcCoeSdoRead.bError
		OR (NOT fbEcGetSlaveName.bBusy
			AND fbEcGetSlaveName.bError)
		THEN
		
			fbEcCoeSdoRead(bExecute := FALSE); 
			fbEcGetSlaveName(bExecute := FALSE); 

		END_IF

	END_IF
	
(* End *)
END_ACTION

ACTION act_Signals:
(* Evaluate the input (EL3214-0090) signals *)

	IF nEcSlaveState.3 (* Slave in operational state *)
	THEN
		(* OP -> transfer the signal states *)
		nInSafeDataValue1 := stInfoData.nInSafeDataValue1;
		nInSafeDataValue2 := stInfoData.nInSafeDataValue2;
		nInSafeDataValue3 := stInfoData.nInSafeDataValue3;
		nInSafeDataValue4 := stInfoData.nInSafeDataValue4;
	ELSE
		(* Error -> clear the signal states *)
		nInSafeDataValue1 := nInSafeDataValue2 := nInSafeDataValue3 := nInSafeDataValue4 := 0;
	END_IF

(* End *)
END_ACTION

END_FUNCTION_BLOCK

// ---- POUs/TwinSAFE/Components/FB_TwinSafeConnectionEL5021.TcPOU
FUNCTION_BLOCK FB_TwinSafeConnectionEL5021
(*******************************************************************************************************
Description			:	Evaluate a TwinSAFE connection status and diagnosis to an EtherCAT terminal
Supported terminals : 	EL5021-0090
Documentation 		:	
Version/Date 		:	
Required libraries 	: 	TcSystem.lib (Tc2_System), TcEtherCAT.lib (Tc2_EtherCAT)
********************************************************************************************************)
VAR_INPUT
END_VAR
VAR_OUTPUT

	stInfoData						AT %I*	:ST_TsConnectionInfoEL5021;		(* EL6900 \ Connection Info Data \ Message_X Info Data*)
	nEcSlaveState					AT %I*	:UINT ;							(* EL5021-0090 \ InfoData \ State *)
	stEcAdsAddr						AT %I*	:ST_AdsAddr;					(* EL5021-0090 \ InfoData \ AdsAddr *)

(* act_EcSlaveIdentify *)
	sEcSlaveType							:STRING(15);
	sEcSlaveName							:STRING(31) := '';
	bSlaveIdentify							:BOOL;
	bSlaveTypeError							:BOOL;
	
(* act_Signals *)
	nInSafeDataCounterValue					:UDINT;
	nInSafeDataFrequencyValue				:DINT;
	nInSafeDataFrequencyValue16Bit			:INT;

(* act_ConnectionState *)
	sState									:STRING;
	
(* act_ConnectionDiag *)
	sDiag									:STRING;
	sFault									:STRING;						(* FailSafe Error (Hardware)*)
	bError									:BOOL;							(* TwinSAFE-Error *)
	
END_VAR
VAR

(* act_ConnectionDiag *)
	nDiag0_3								:BYTE;

(* act_EcSlaveIdentify *)
	fbEcCoeSdoRead							:FB_EcCoESdoReadEx;
	fbEcGetSlaveName						:FB_EcGetSlaveName;

END_VAR
(* End *)

(* Function Block TwinSAFE connection status and diagnosis for EL1904 Terminals *)

(* THIS CODE IS ONLY AN EXAMPLE - YOU HAVE TO CHECK APTITUDE FOR YOUR APPLICATION *)

	(* Identify the EtherCAT slave *)
		act_EcSlaveIdentify();

	(* Evaluate the connection state *)
		act_ConnectionState();
	
	(* Evaluate the connection diagnosis *)
		act_ConnectionDiag();
	
	(* Evaluate the EL1904 input signals *)
		act_Signals();
	
(* End *)

ACTION act_ConnectionDiag:
(* Evaluate the connection diagnosis *)

	(* Evaluate Bit 0..3 *)
	nDiag0_3 := USINT_TO_BYTE(stInfoData.nDiag) AND 16#0F;

	CASE nDiag0_3 OF
		0:		sDiag := 'No error';
		1:		sDiag := 'Invalid command';
		2:		sDiag := 'Unknown command';
		3:		sDiag := 'Invalid connection ID';
		4:		sDiag := 'Invalid CRC';
		5:		sDiag := 'Watchdog time elapsed';
		6:		sDiag := 'Invalid FSOE address';
		7:		sDiag := 'Invalid data';
		8:		sDiag := 'Invalid communication parameter length';
		9:		sDiag := 'Invalid communication parameters';
		10:		sDiag := 'Invalid user parameter length';
		11:		sDiag := 'Invalid user parameter';
		12:		sDiag := 'FSoE master reset';
		13:		sDiag := 'Module err detected on slave, with option "Module error is ComError" activated';
		14:		sDiag := 'Module err detected on EL290x, with option "Error acknowledge active" activated';
		15:		sDiag := 'Slave not yet started, or unexpected error argument';
	END_CASE

	(* Evaluate Bit 4..7 *)
	sFault:='';

	IF stInfoData.nDiag.4 
	THEN
		sFault	:= 'FSoE slave error detected - '; 
	END_IF

	IF stInfoData.nDiag.5 
	THEN
		sFault	:= concat(sFault,'FSoE slave reports Failsafe Value active - ');
	END_IF

	IF stInfoData.nDiag.6 
	THEN
		sFault	:= concat(sFault,'StartUp - ');
	END_IF

	IF stInfoData.nDiag.7 
	THEN
		sFault	:= concat(sFault, 'FSoE master reports Failsafe Value active');
	END_IF
		
	(* Error *)
	bError := stInfoData.nDiag <> 0;

(* End *)
END_ACTION

ACTION act_ConnectionState:
(* Evaluate the connection state *)

	CASE stInfoData.nState OF
		100:	sState := 'Reset state';
		101:	sState := 'Session state';
		102:	sState := 'Connection state';
		103:	sState := 'Parameter state';
		104:	sState := 'Data state';
		105:	sState := 'Shutdown state';
	ELSE
		sState := 'unknown';
	END_CASE
	
(* End *)
END_ACTION

ACTION act_EcSlaveIdentify:
(* Identify the EtherCAT slave *)

	IF NOT nEcSlaveState.3
	THEN
		bSlaveIdentify  := FALSE;
		bSlaveTypeError := FALSE;
		sEcSlaveType    := '';
	END_IF

	IF nEcSlaveState.3
		AND NOT bSlaveIdentify
		AND NOT bSlaveTypeError
 		AND F_CreateAmsNetId(stEcAdsAddr.netId) <> '0.0.0.0.0.0' 
		AND stEcAdsAddr.port <> 0
	THEN

		fbEcCoeSdoRead(
			sNetId			:= 	F_CreateAmsNetId(stEcAdsAddr.netId),
			nSlaveAddr		:= 	stEcAdsAddr.port,
			nSubIndex		:= 	0,
			nIndex			:= 	16#1008,
			pDstBuf			:= 	ADR(sEcSlaveType),
			cbBufLen		:= 	SIZEOF(sEcSlaveType),
			bExecute		:= 	TRUE,
			tTimeout		:= 	DEFAULT_ADS_TIMEOUT);
	

		fbEcGetSlaveName(
			bExecute		:=	TRUE, 
			sNetId			:=	F_CreateAmsNetId(stEcAdsAddr.netId), 
			nSlaveAddr		:=	stEcAdsAddr.port, 
			tTimeout		:=	DEFAULT_ADS_TIMEOUT, 
			bBusy			=>	, 
			sSlaveName		=>	sEcSlaveName, 
			bError			=>	, 
			nErrId			=>	);

		IF NOT fbEcCoeSdoRead.bBusy
			AND NOT fbEcCoeSdoRead.bError
			AND NOT fbEcGetSlaveName.bBusy
			AND NOT fbEcGetSlaveName.bError
		THEN
		
			fbEcCoeSdoRead(bExecute := FALSE); 
			fbEcGetSlaveName(bExecute := FALSE); 

			IF sEcSlaveType = 'EL5021-0090' 
				AND fbEcGetSlaveName.sSlaveName <> ''
			THEN
				bSlaveIdentify := TRUE;
			ELSE
				bSlaveTypeError := TRUE;
			END_IF

		ELSIF NOT fbEcCoeSdoRead.bBusy
			AND fbEcCoeSdoRead.bError
		OR (NOT fbEcGetSlaveName.bBusy
			AND fbEcGetSlaveName.bError)
		THEN
		
			fbEcCoeSdoRead(bExecute := FALSE); 
			fbEcGetSlaveName(bExecute := FALSE); 

		END_IF

	END_IF
	
(* End *)
END_ACTION

ACTION act_Signals:
(* Evaluate the input (EL5021-0090) signals *)

	IF nEcSlaveState.3 (* Slave in operational state *)
	THEN
		(* OP -> transfer the signal states *)
		nInSafeDataCounterValue			:= stInfoData.nInSafeDataCounterValue;			
		nInSafeDataFrequencyValue		:= stInfoData.nInSafeDataFrequencyValue;
		nInSafeDataFrequencyValue16Bit	:= stInfoData.nInSafeDataFrequencyValue16Bit;
	ELSE
		(* Error -> clear the signal states *)
		nInSafeDataCounterValue 	   := 0;
		nInSafeDataFrequencyValue 	   := 0; 
		nInSafeDataFrequencyValue16Bit := 0;
	END_IF

(* End *)
END_ACTION

END_FUNCTION_BLOCK

// ---- POUs/TwinSAFE/Components/FB_TwinSafeGroupExt.TcPOU
FUNCTION_BLOCK FB_TwinSafeGroupExt
(*******************************************************************************************************
Description			:	Entries of the status and diagnostic TwinSAFE groups
ocumentation 		:	TwinSAFE-Logik-FB TwinCAT function blocks for TwinSAFE logic terminals
Supported hardware	: 	EL6910 / EJ6910 / EK1960
Version/Date 		:	V3.1.0/26.10.2016
********************************************************************************************************)
VAR_INPUT

	bRun							AT %Q*	:BOOL;				(* TwinSAFE group run - linked with the associated TwinSAFE Group in the TwinSAFE projekt *)
	bErrAck							AT %Q*	:BOOL;				(* TwinSAFE group error acknowledge - linked with the associated TwinSAFE Group in the TwinSAFE projekt *)
	bModuleFault					AT %Q*	:BOOL;				(*  *)
	sName									:STRING;			(* TwinSAFE group name *)

END_VAR
VAR_OUTPUT

	stInfoData						AT %I*	:ST_TsGroupInfo;	(* TwinSAFE Group Info Data *)
	bComErr							AT %I*	:BOOL;				(* TwinSAFE group communication error - linked with the associated TwinSAFE Group in the TwinSAFE projekt *)
	bFbErr							AT %I*	:BOOL;				(* TwinSAFE group function block error - linked with the associated TwinSAFE Group in the TwinSAFE projekt *)
	bOutErr							AT %I*	:BOOL;				(* TwinSAFE group output error - linked with the associated TwinSAFE Group in the TwinSAFE projekt *)
	bOtherErr						AT %I*	:BOOL;				(* ModuleFault or AnalogValueFault or WaitComTimeoutFault *)
	bComStartUp						AT %I*	:BOOL;				(* At least one of the Connection of this group is in the StartUp *)
	bFbDeactive						AT %I*	:BOOL;				(* TwinSAFE group was deactivated *)
	bFbRun							AT %I*	:BOOL;				(* All Fbs are in run state *)
	bInRun							AT %I*	:BOOL;				(* TwinSAFE group is in run *)
	sState									:STRING;
	sDiag									:STRING;

END_VAR
VAR
END_VAR
(* End *)

(* TwinSAFE group status and diagnostic *)

(* THIS CODE IS ONLY AN EXAMPLE - YOU HAVE TO CHECK APTITUDE FOR YOUR APPLICATION *)

	CASE stInfoData.nState OF
		1:	sState := 'RUN';
		2:	sState := 'STOP';
		4:	sState := 'ERROR';
		5:	sState := 'RESET';
		6:	sState := 'START';
		7:	sState := 'STOPERROR';
		16:	sState := 'DEACTIVE';
		17:	sState := 'WAITCOMERROR';
	ELSE
		sState := 'undefined';
	END_CASE
	
	CASE stInfoData.nDiag OF
		0:	sDiag := 'No error';
		1:	sDiag := 'Fb error';
		2:	sDiag := 'Com error';
		3:	sDiag := 'Module error';
		4:	sDiag := 'CMP error';
		5:	sDiag := 'Deactivate error';
		6:	sDiag := 'Restart error';
	ELSE
		sDiag := 'undefined';
	END_CASE
	
(* End *)

END_FUNCTION_BLOCK

// ---- POUs/Sample OOP Conveyor/Axis Blocks/FB_Stepper.TcPOU
FUNCTION_BLOCK FB_Stepper EXTENDS FB_AxisNc
VAR_INPUT
	nStatusByte : BYTE;
END_VAR
VAR_OUTPUT
	nCtrlByte : BYTE; 
END_VAR
VAR
END_VAR

METHOD PUBLIC M_HardwareReset : UDINT
//Set bit 6 in the Control word that will be transmitted to the stepper for resetting. 
VAR_INPUT
	bReset : BOOL;
END_VAR
//REturn 0 when idle
//Return 1 when busy 
//return 3 when complete
VAR_INST // added by the converter: edge detectors and wires of the graphical bodies
    _w1, _w2 : BOOL;
    _w3, _w4 : ANY;
END_VAR
_w1 := bReset;
IF _w1 THEN (* 1; result not used *) END_IF
M_HardwareReset := _w1;
IF _w2 THEN _w3 := 0; END_IF
_w2 := NOT bReset;
M_HardwareReset := _w3;
IF bReset THEN _w4 := 1; END_IF
nCtrlByte.6 := _w4;
END_METHOD

END_FUNCTION_BLOCK

// ---- GlobalTextList.TcGTLO
TEXTLIST GlobalTextList
  48 = '\n\nS33'
  32 = '\n\n\nS10'
  33 = '\n\n\nTest'
  35 = '\n\nS10'
  39 = '\n\nS30'
  37 = '\n\nS31'
  44 = '\n\nS32'
  45 = '\n\nS33'
  34 = '\n\nTest'
  51 = '\nS10'
  52 = '\nS11'
  53 = '\nS12'
  54 = '\nS13'
  55 = '\nS14'
  56 = '\nS15'
  57 = '\nS16'
  58 = '\nS17'
  59 = '\nS20'
  60 = '\nS21'
  61 = '\nS22'
  62 = '\nS23'
  63 = '\nS24'
  64 = '\nS25'
  65 = '\nS26'
  66 = '\nS27'
  118 = '\nS30'
  38 = '\nS31'
  47 = '\nS32'
  50 = '\nS33'
  46 = '\nTest'
  109 = '                                               '
  110 = '                                                            '
  112 = '                                                              '
  111 = '                                                               '
  100 = '    Axis 1 - EL7037 - AS1020-0120    '
  101 = '  Axis 1 - EL7037 - AS1020-0120    '
  1438 = ' Actual Motion Sample Mode: %s'
  102 = ' Axis 1 - EL7037 - AS1020-0120      '
  103 = ' Axis 2 - EL7201 - AM8111-0F20      '
  104 = ' Axis 3 - AX5203-A - AM8111-0F10      '
  105 = ' Axis 4 - AX5203-B - AM8111-0F21      '
  1444 = ' MC2-Sample Mode: %s'
  1450 = ' NCI-Sample Mode: %s'
  1467 = ' OOP-Conveyor-Sample Mode: %s'
  1461 = ' OOP-Sample Mode: %s'
  966 = ' Reversing'
  1455 = ' Sample Mode Request'
  127 = '%.2f'
  97 = '%.3d'
  68 = '%.3f'
  71 = '%.3f  '
  86 = '%.3f    '
  70 = '%.3f Degree'
  942 = '%1.3f'
  91 = '%d'
  98 = '%d   '
  173 = '%d    '
  114 = '%d         '
  113 = '%d   .'
  116 = '%d INC '
  117 = '%d INC     '
  115 = '%d----'
  4 = '%s'
  14 = '%s ComErr'
  15 = '%s FbErr'
  607 = '0'
  609 = '1'
  611 = '2'
  613 = '3'
  615 = '4'
  617 = '5'
  156 = 'A\nX\nI\nS\n1'
  157 = 'A\nX\nI\nS\n2'
  959 = 'Absolute'
  77 = 'Absolute position:'
  119 = 'Absolute target position:'
  2958 = 'Accel'
  1992 = 'Act'
  1541 = 'Add SIN Wabe'
  1244 = 'Add SIN Wave'
  0 = 'Addr'
  2929 = 'Amplitude'
  89 = 'Analog'
  90 = 'Analog / Handwheel'
  43 = 'Analog Box'
  2909 = 'Angle'
  171 = 'AXIS'
  175 = 'Axis'
  178 = 'AXIS\nSEQUENCE'
  69 = 'Axis 1'
  73 = 'Axis 1 (AS1020-0120)'
  74 = 'Axis 1 - EL7037 - AS1020-0120'
  99 = 'Axis 1 EL7037 AS1020-0120'
  83 = 'Axis 2 - EL7201 - AM8111-0F20'
  84 = 'Axis 3 - AX5203-A - AM8111-0F10'
  85 = 'Axis 4 - AX5203-B - AM8111-0F21'
  67 = 'Axis Box'
  176 = 'Axis Ref.'
  169 = 'Axis reversing\nsequence'
  177 = 'Axis Sequence'
  209 = 'AXIS SEQUENCE'
  1052 = 'Axis State'
  945 = 'Axis1/Master'
  948 = 'Axis2/Slave'
  170 = 'AXISREVERSING'
  208 = 'AXISSEQUENCE'
  108 = 'AxisStatusOverview.sGroupName'
  1545 = 'bAllInfoCopiedToFile'
  1531 = 'bInitFinished'
  2348 = 'bPenDown'
  1559 = 'bSendToClientFinished'
  1552 = 'bSendToMasterFinished'
  2620 = 'Bufferd_SuprImposed'
  1100 = 'Buffered and Superimposed'
  2621 = 'Buffered and Superimposed Moves'
  219 = 'Buffered Move'
  2099 = 'Buffered_Superimposed'
  1538 = 'bUseXmlFormat'
  146 = 'C-Err\nAck'
  136 = 'C-h1'
  147 = 'C-SDIn'
  148 = 'C-SDIp'
  152 = 'C-SMM1'
  150 = 'C-SOS1'
  154 = 'C-SS1'
  155 = 'C-SS2'
  151 = 'C-SSM2'
  149 = 'C-SSR1'
  153 = 'C-STO'
  2489 = 'Cam IN'
  220 = 'CAM In'
  2505 = 'Cam OUT'
  221 = 'CAM Out'
  629 = 'CAM out and re-init required'
  2122 = 'Cam Table'
  931 = 'Camming_ MotnFns'
  928 = 'CamTable'
  5 = 'Ch1'
  131 = 'Ch1\n'
  202 = 'Ch1\n%d\nINC'
  197 = 'Ch1In'
  199 = 'Ch1Out'
  6 = 'Ch2'
  203 = 'Ch2\n%d\nINC'
  198 = 'Ch2In'
  200 = 'Ch2Out'
  7 = 'Ch3'
  204 = 'Ch3\n%d\nINC'
  8 = 'Ch4'
  205 = 'Ch4\n%d\nINC'
  164 = 'Com Err'
  163 = 'Com Error'
  160 = 'ComErr'
  2125 = 'Command Speed : %4.2f'
  212 = 'Conveyor 1'
  213 = 'Conveyor 2'
  214 = 'Conveyor 3'
  1106 = 'Counter OFF:  %d'
  1101 = 'Counter ON:  %d'
  206 = 'Counter Value:\n%d\nINC'
  124 = 'Coupelt'
  125 = 'Coupled'
  72 = 'Degree'
  126 = 'Degree/s'
  9 = 'Diag: %s'
  1566 = 'DO counter: %i'
  1307 = 'Dynamic Gearing'
  79 = 'Enable'
  1580 = 'ENTRY counter: %i'
  132 = 'Err'
  159 = 'Err Ack'
  201 = 'Err Cc'
  133 = 'Err Es or Cc'
  135 = 'Err input pair'
  134 = 'Err Ol or Cv'
  78 = 'Error'
  81 = 'Error : %d'
  1539 = 'Error Ack'
  82 = 'Error Id: %d'
  27 = 'EtherCAT\nDIAGNOSTIC'
  207 = 'EtherCAT DIAGNOSTIC'
  1573 = 'EXIT counter: %i'
  1056 = 'Expired Time of Sample'
  872 = 'Ext SP Gen Enable'
  2880 = 'Ext SP Gen OFF'
  2871 = 'Ext SP Gen ON'
  571 = 'External Setpoint Generator'
  935 = 'External_SP_Gen'
  161 = 'Fb Err'
  162 = 'Fb Error'
  26 = 'fdsaasd'
  1312 = 'Flying Saw'
  1498 = 'FlyingSaw_Gearing'
  753 = 'Frequency'
  2382 = 'Gcode file to execute:'
  924 = 'Gearing_FlyingSaw'
  25 = 'Group 1'
  1314 = 'GroupBox'
  107 = 'Hallo'
  96 = 'Handwheel S18:'
  1620 = 'ID %d'
  174 = 'Idle Time:'
  2938 = 'Increment/frequency'
  92 = 'Increments'
  2198 = 'Infeed Conveyor'
  2473 = 'Init CAM Table'
  738 = 'InitState'
  2465 = 'Interpolation Type'
  1997 = 'Jog Bwd'
  1988 = 'Jog Fwd'
  2373 = 'Last 10 executed Gcode blocks'
  2904 = 'Last 5 executed Gcode blocks'
  621 = 'Linear'
  619 = 'Load Points'
  2225 = 'Machine Operation\n1. Switch to Auto\n2 Press the Run Conveyor Button\n3. Put Part On Infeed will prepare a \npart to be loaded.\n3. Press all pick and place buttons for\n automatic part transferrring\n\nWhen a part reaches the Pick Pos\nIt will be picked and placed on the\nthe next conveyor. \nIt will leave the system when it reaches \nthe end of the outfeed conveyor\nFor Full Documentation open the \nDocument.PDF it is the first item in \nthe POU list in the solution explorer'
  211 = 'Machine State %s'
  2380 = 'Master'
  2372 = 'Master Pos at Trigger'
  1847 = 'MasterPos'
  76 = 'Modulo position:'
  856 = 'MOTION PROFILES'
  610 = 'MOTION SEQUENCE'
  952 = 'Move'
  172 = 'ms'
  1 = 'Name'
  938 = 'NCI'
  2365 = 'NCI ErrId'
  2385 = 'NCI Error ID:'
  2357 = 'NCI State'
  2669 = 'NCI State:'
  1303 = 'No Gearing'
  2513 = 'not Periodic'
  574 = 'Not Periodic'
  2216 = 'Outfeed Conveyor'
  216 = 'Part ID To Place %d'
  2497 = 'Periodic'
  1640 = 'Pick Part'
  1627 = 'Pick Pos: %4.2f'
  1654 = 'Place Part'
  1841 = 'Point'
  627 = 'Point to change'
  784 = 'Pos %4.2f'
  969 = 'Pos / Dist'
  2948 = 'Position'
  75 = 'Position absolute:'
  95 = 'Potentiometer R10:'
  93 = 'Potentiometer R11 position:'
  94 = 'Potentiometer R11:'
  2610 = 'Power'
  752 = 'PublishToClient'
  749 = 'PublishToMaster'
  215 = 'Put Part On Infeed'
  122 = 'R'
  1484 = 'Read Points\nFrom File'
  80 = 'Reference cam'
  962 = 'Relative'
  2481 = 'relative slave motion'
  1060 = 'Remaining Time for Sample'
  196 = 'Reset'
  1501 = 'REVERSEING SEQUENCE'
  1991 = 'REVERSING SEQUENCE'
  158 = 'Run'
  2803 = 'Run NCI'
  145 = 'S-Err\nAck'
  144 = 'S-SDIn'
  143 = 'S-SDIp'
  138 = 'S-SMM1'
  141 = 'S-SOS1'
  140 = 'S-SSM2'
  142 = 'S-SSR1'
  137 = 'S-STO'
  139 = 'S/SMM1'
  31 = 'S10'
  180 = 'S11'
  181 = 'S12'
  182 = 'S13'
  183 = 'S14'
  184 = 'S15'
  185 = 'S16'
  186 = 'S17'
  188 = 'S20'
  189 = 'S21'
  190 = 'S22'
  191 = 'S23'
  192 = 'S24'
  193 = 'S25'
  194 = 'S26'
  195 = 'S27'
  179 = 'S30'
  36 = 'S31'
  187 = 'S32'
  49 = 'S33'
  1985 = 'Set'
  106 = 'sGroupName'
  1138 = 'SIN Wave Gen Enable'
  2900 = 'SIN Wave Gen OFF'
  2890 = 'SIN Wave Gen ON'
  2919 = 'SinWave'
  2388 = 'Slave'
  2396 = 'Slave Gear Ratio'
  1853 = 'SlavePos'
  1858 = 'SlaveVelo'
  625 = 'Sliding Spline'
  1634 = 'Spacing: %4.2f'
  2135 = 'Speed : %4.2f'
  1979 = 'Speed : %f'
  623 = 'Spline'
  120 = 'Start'
  29 = 'Start Page'
  30 = 'START PAGE'
  10 = 'State: %s'
  3 = 'Status'
  123 = 'Stop'
  218 = 'SuperImposed Distance'
  2124 = 'Superimposed Distance'
  217 = 'SuperImposed Move'
  1481 = 'Superimposed Move'
  87 = 'Switch'
  41 = 'Switch Box'
  1661 = 'Switch To Auto'
  1667 = 'Switch To Manual'
  88 = 'Switches'
  1316 = 'Sync Positions'
  11 = 'T1 %s'
  16 = 'T1 %s °C'
  18 = 'T1: %s °C'
  12 = 'T2 %s'
  17 = 'T2 %s °C'
  19 = 'T2: %s °C'
  1202 = 'Target Distance'
  2988 = 'Target Distance2'
  165 = 'Target position 1:'
  167 = 'Target position 2:'
  129 = 'Target position:'
  3154 = 'Target Velocity'
  166 = 'Target velocity 1:'
  168 = 'Target velocity 2:'
  2997 = 'Target Velocity2'
  128 = 'Target velocity:'
  121 = 'Test'
  745 = 'TextFormat'
  130 = 'TO: %s °C'
  2207 = 'Transfer Conveyor 2 to Outfeed'
  1633 = 'Transfer Infeed to Conveyor 2'
  1647 = 'Transfer Part ID %d'
  40 = 'TwinSAFE'
  28 = 'TwinSAFE\nDIAGNOSTIC'
  42 = 'TwinSAFE Box'
  21 = 'TwinSAFE connection diagnostic'
  210 = 'TwinSAFE DIAGNOSTIC'
  24 = 'TwinSAFE function block diagnostic'
  23 = 'TwinSAFE function blocks diagnostic'
  20 = 'TwinSAFE group diagnostic'
  22 = 'TwinSAFE terminal connection diagnostic'
  13 = 'Typ: %s'
  2 = 'Type'
  973 = 'Velocity'
  742 = 'XmlFormat'
  955 = 'Zero'
END_TEXTLIST

// ---- POUs/MainPOUs/V_MAIN.TcVIS
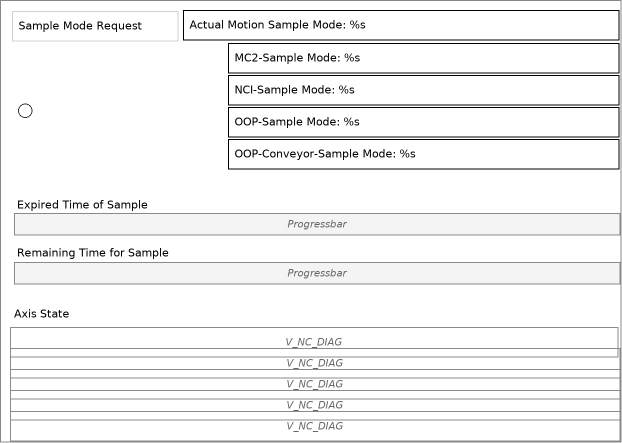
VISUALIZATION V_MAIN  // 622x443
    Rectangle (183,10 436x30), "Actual Motion Sample Mode: %s", text variable: MAIN.eSampleMode
    Rectangle (228,43 391x30), "MC2-Sample Mode: %s", text variable: MAIN.eSampleModeMC2, colour toggle: MAIN.eSampleMode = eSMode_MC2_Req
    Rectangle (228,75 391x30), "NCI-Sample Mode: %s", text variable: MAIN.eSampleModeNCI, colour toggle: MAIN.eSampleMode = eSMode_NCI_Req
    RadioButton (16,46 131x129), variable: MAIN.nRadioButton
        Areas[0]: Text=Idle
        Areas[4]: Text=OOP Convyor
    Textfield (12,11 166x30), "Sample Mode Request"
    Rectangle (228,107 391x30), "OOP-Sample Mode: %s", text variable: MAIN.eSampleModeOOP, colour toggle: MAIN.eSampleMode = eSMode_OOP_Req
    Rectangle (228,139 391x30), "OOP-Conveyor-Sample Mode: %s", text variable: MAIN.eSampleModeOOPConv, colour toggle: MAIN.eSampleMode = eSMode_OOPConv_Req
    Frame (10,327 608x30)
        shows V_NC_DIAG(AxisRef := MAIN.AxisRef[1])
    Frame (10,348 610x30)
        shows V_NC_DIAG(AxisRef := MAIN.AxisRef[2])
    Frame (10,369 610x30)
        shows V_NC_DIAG(AxisRef := MAIN.AxisRef[3])
    Frame (10,390 610x30)
        shows V_NC_DIAG(AxisRef := MAIN.AxisRef[4])
    Frame (10,411 610x30)
        shows V_NC_DIAG(AxisRef := MAIN.AxisRef[5])
    Progressbar (14,213 606x22), variable: 60-MAIN.nRemainingModeTime
    Progressbar (14,262 606x22), variable: MAIN.nRemainingModeTime
    Label (11,299 150x30), "Axis State"
    Label (14,190 150x30), "Expired Time of Sample"
    Label (14,238 225x30), "Remaining Time for Sample"
END_VISUALIZATION

// ---- POUs/Sample OOP Conveyor/Internal Visus/Conveyor.TcVIS
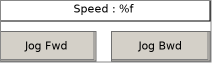
VISUALIZATION Conveyor  // 212x63
VAR_IN_OUT
	bJogFwd: BOOL;
	bJogBwd: BOOL;
	fSpeed: LREAL;
END_VAR
    Rectangle (-3,-3 213x24), "Speed : %f", text variable: fSpeed
    Button (-3,31 99x30), "Jog Fwd"
        tap bJogFwd
    Button (111,31 99x30), "Jog Bwd"
        tap bJogBwd
END_VISUALIZATION

// ---- POUs/Sample OOP Conveyor/Internal Visus/ConveyorAuto.TcVIS
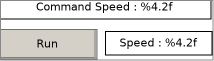
VISUALIZATION ConveyorAuto  // 214x61
VAR_IN_OUT
	bRunConveyor : BOOL;
	fActualSpeed : LREAL;
	fCmdSpeed : LREAL;
END_VAR
    Rectangle (-2,-5 213x24), "Command Speed : %4.2f", text variable: fCmdSpeed
        OnMouseClick: write fCmdSpeed via Edit, min 1, max 2000
    Button (-2,29 99x30), "Run"
        toggle bRunConveyor
    Rectangle (105,31 107x24), "Speed : %4.2f", text variable: fActualSpeed
END_VISUALIZATION

// ---- POUs/Sample OOP Conveyor/Internal Visus/ConveyorData.TcVIS
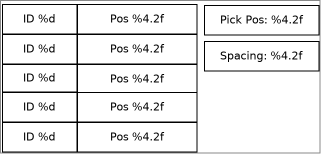
VISUALIZATION ConveyorData  // 321x154
VAR_IN_OUT
	fbConveyor : FB_Conveyor;
END_VAR
    Rectangle (77,4 120x30), "Pos %4.2f", text variable: fbConveyor.arrProductsOnConveyor[1].fPosition
    Rectangle (77,34 120x30), "Pos %4.2f", text variable: fbConveyor.arrProductsOnConveyor[2].fPosition
    Rectangle (77,64 120x30), "Pos %4.2f", text variable: fbConveyor.arrProductsOnConveyor[3].fPosition
    Rectangle (77,92 120x30), "Pos %4.2f", text variable: fbConveyor.arrProductsOnConveyor[4].fPosition
    Rectangle (77,122 120x30), "Pos %4.2f", text variable: fbConveyor.arrProductsOnConveyor[5].fPosition
    Rectangle (2,4 75x30), "ID %d", text variable: fbConveyor.arrProductsOnConveyor[1].iIDNumber
    Rectangle (2,34 75x30), "ID %d", text variable: fbConveyor.arrProductsOnConveyor[2].iIDNumber
    Rectangle (2,64 75x28), "ID %d", text variable: fbConveyor.arrProductsOnConveyor[3].iIDNumber
    Rectangle (2,92 75x30), "ID %d", text variable: fbConveyor.arrProductsOnConveyor[4].iIDNumber
    Rectangle (2,122 75x30), "ID %d", text variable: fbConveyor.arrProductsOnConveyor[5].iIDNumber
    Rectangle (204,5 115x30), "Pick Pos: %4.2f", text variable: fbConveyor.fPickLocation
    Rectangle (204,41 115x30), "Spacing: %4.2f", text variable: fbConveyor.fMinimumSpacing
END_VISUALIZATION

// ---- POUs/Sample OOP Conveyor/V_OOP_Conveyor.TcVIS
